gfCNCPoint3[21625] = {X 108.1088, Y 46.8612, Z -4.6667, A 0.000, B 0.000, C 0.000 }
gfCNCPoint3[21626] = {X 107.7913, Y 45.9714, Z -4.6667, A 0.000, B 0.000, C 0.000 }
gfCNCPoint3[21627] = {X 107.6786, Y 45.0335, Z -4.6667, A 0.000, B 0.000, C 0.000 }
gfCNCPoint3[21628] = {X 107.6785, Y 44.1775, Z -4.6667, A 0.000, B 0.000, C 0.000 }
gfCNCPoint3[21629] = {X 107.7133, Y 43.6465, Z -4.6667, A 0.000, B 0.000, C 0.000 }
gfCNCPoint3[21630] = {X 107.8171, Y 43.1246, Z -4.6667, A 0.000, B 0.000, C 0.000 }
gfCNCPoint3[21631] = {X 107.9815, Y 42.6369, Z -4.6667, A 0.000, B 0.000, C 0.000 }
gfCNCPoint3[21632] = {X 108.2062, Y 42.1739, Z -4.6667, A 0.000, B 0.000, C 0.000 }
gfCNCPoint3[21633] = {X 108.6606, Y 41.4995, Z -4.6667, A 0.000, B 0.000, C 0.000 }
gfCNCPoint3[21634] = {X 109.2059, Y 40.8963, Z -4.6667, A 0.000, B 0.000, C 0.000 }
gfCNCPoint3[21635] = {X 109.2058, Y 39.1629, Z -4.6667, A 0.000, B 0.000, C 0.000 }
gfCNCPoint3[21636] = {X 109.0939, Y 39.1629, Z -4.6667, A 0.000, B 0.000, C 0.000 }
gfCNCPoint3[21637] = {X 106.0379, Y 46.6307, Z -4.6667, A 0.000, B 0.000, C 0.000 }
gfCNCPoint3[21638] = {X 105.6747, Y 47.3174, Z -4.6667, A 0.000, B 0.000, C 0.000 }
gfCNCPoint3[21639] = {X 105.1923, Y 47.9263, Z -4.6667, A 0.000, B 0.000, C 0.000 }
gfCNCPoint3[21640] = {X 104.6069, Y 48.4370, Z -4.6667, A 0.000, B 0.000, C 0.000 }
gfCNCPoint3[21641] = {X 103.9382, Y 48.8323, Z -4.6667, A 0.000, B 0.000, C 0.000 }
gfCNCPoint3[21642] = {X 103.0119, Y 49.1460, Z -4.6667, A 0.000, B 0.000, C 0.000 }
gfCNCPoint3[21643] = {X 102.0384, Y 49.2391, Z -4.6667, A 0.000, B 0.000, C 0.000 }
gfCNCPoint3[21644] = {X 101.0695, Y 49.1068, Z -4.6667, A 0.000, B 0.000, C 0.000 }
gfCNCPoint3[21645] = {X 100.1566, Y 48.7559, Z -4.6667, A 0.000, B 0.000, C 0.000 }
gfCNCPoint3[21646] = {X 99.3484, Y 48.2052, Z -4.6667, A 0.000, B 0.000, C 0.000 }
gfCNCPoint3[21647] = {X 98.6879, Y 47.4840, Z -4.6667, A 0.000, B 0.000, C 0.000 }
gfCNCPoint3[21648] = {X 98.2102, Y 46.6307, Z -4.6667, A 0.000, B 0.000, C 0.000 }
gfCNCPoint3[21649] = {X 95.0510, Y 38.9046, Z -4.6667, A 0.000, B 0.000, C 0.000 }
gfCNCPoint3[21650] = {X 95.0511, Y 40.9419, Z -4.6667, A 0.000, B 0.000, C 0.000 }
gfCNCPoint3[21651] = {X 95.5851, Y 41.4821, Z -4.6667, A 0.000, B 0.000, C 0.000 }
gfCNCPoint3[21652] = {X 96.0162, Y 42.1073, Z -4.6667, A 0.000, B 0.000, C 0.000 }
gfCNCPoint3[21653] = {X 96.2570, Y 42.6034, Z -4.6667, A 0.000, B 0.000, C 0.000 }
gfCNCPoint3[21654] = {X 96.4328, Y 43.1260, Z -4.6667, A 0.000, B 0.000, C 0.000 }
gfCNCPoint3[21655] = {X 96.5399, Y 43.6619, Z -4.6667, A 0.000, B 0.000, C 0.000 }
gfCNCPoint3[21656] = {X 96.5785, Y 44.2071, Z -4.6667, A 0.000, B 0.000, C 0.000 }
gfCNCPoint3[21657] = {X 96.5783, Y 45.0408, Z -4.6667, A 0.000, B 0.000, C 0.000 }
gfCNCPoint3[21658] = {X 96.4643, Y 45.9775, Z -4.6667, A 0.000, B 0.000, C 0.000 }
gfCNCPoint3[21659] = {X 96.1459, Y 46.8659, Z -4.6667, A 0.000, B 0.000, C 0.000 }
gfCNCPoint3[21660] = {X 95.6389, Y 47.6618, Z -4.6667, A 0.000, B 0.000, C 0.000 }
gfCNCPoint3[21661] = {X 94.9685, Y 48.3258, Z -4.6667, A 0.000, B 0.000, C 0.000 }
gfCNCPoint3[21662] = {X 94.1677, Y 48.8251, Z -4.6667, A 0.000, B 0.000, C 0.000 }
gfCNCPoint3[21663] = {X 93.2764, Y 49.1350, Z -4.6667, A 0.000, B 0.000, C 0.000 }
gfCNCPoint3[21664] = {X 92.3385, Y 49.2400, Z -4.6667, A 0.000, B 0.000, C 0.000 }
gfCNCPoint3[21665] = {X 85.8951, Y 49.2400, Z -4.6667, A 0.000, B 0.000, C 0.000 }
gfCNCPoint3[21666] = {X 84.9564, Y 49.1348, Z -4.6667, A 0.000, B 0.000, C 0.000 }
gfCNCPoint3[21667] = {X 84.0643, Y 48.8244, Z -4.6667, A 0.000, B 0.000, C 0.000 }
gfCNCPoint3[21668] = {X 83.2631, Y 48.3242, Z -4.6667, A 0.000, B 0.000, C 0.000 }
gfCNCPoint3[21669] = {X 82.5924, Y 47.6590, Z -4.6667, A 0.000, B 0.000, C 0.000 }
gfCNCPoint3[21670] = {X 82.0857, Y 46.8618, Z -4.6667, A 0.000, B 0.000, C 0.000 }
gfCNCPoint3[21671] = {X 81.7681, Y 45.9723, Z -4.6667, A 0.000, B 0.000, C 0.000 }
gfCNCPoint3[21672] = {X 81.6552, Y 45.0345, Z -4.6667, A 0.000, B 0.000, C 0.000 }
gfCNCPoint3[21673] = {X 81.6551, Y 44.2075, Z -4.6667, A 0.000, B 0.000, C 0.000 }
gfCNCPoint3[21674] = {X 81.7604, Y 43.2862, Z -4.6667, A 0.000, B 0.000, C 0.000 }
gfCNCPoint3[21675] = {X 82.0609, Y 42.4090, Z -4.6667, A 0.000, B 0.000, C 0.000 }
gfCNCPoint3[21676] = {X 82.5425, Y 41.6167, Z -4.6667, A 0.000, B 0.000, C 0.000 }
gfCNCPoint3[21677] = {X 83.1828, Y 40.9460, Z -4.6667, A 0.000, B 0.000, C 0.000 }
gfCNCPoint3[21678] = {X 83.1826, Y 28.5916, Z -4.6667, A 0.000, B 0.000, C 0.000 }
gfCNCPoint3[21679] = {X 79.1826, Y 28.5916, Z -4.6667, A 0.000, B 0.000, C 0.000 }
gfCNCPoint3[21680] = {X 83.2626, Y 28.5916, Z -4.6667, A 0.000, B 0.000, C 0.000 }
gfCNCPoint3[21681] = {X 83.2625, Y 16.1991, Z -4.6667, A 0.000, B 0.000, C 0.000 }
gfCNCPoint3[21682] = {X 82.6249, Y 15.5494, Z -4.6667, A 0.000, B 0.000, C 0.000 }
gfCNCPoint3[21683] = {X 82.1439, Y 14.7765, Z -4.6667, A 0.000, B 0.000, C 0.000 }
gfCNCPoint3[21684] = {X 81.8426, Y 13.9176, Z -4.6667, A 0.000, B 0.000, C 0.000 }
gfCNCPoint3[21685] = {X 81.7352, Y 13.0136, Z -4.6667, A 0.000, B 0.000, C 0.000 }
gfCNCPoint3[21686] = {X 81.7351, Y 12.1868, Z -4.6667, A 0.000, B 0.000, C 0.000 }
gfCNCPoint3[21687] = {X 81.8394, Y 11.2611, Z -4.6667, A 0.000, B 0.000, C 0.000 }
gfCNCPoint3[21688] = {X 82.1470, Y 10.3819, Z -4.6667, A 0.000, B 0.000, C 0.000 }
gfCNCPoint3[21689] = {X 82.6427, Y 9.5931, Z -4.6667, A 0.000, B 0.000, C 0.000 }
gfCNCPoint3[21690] = {X 83.3014, Y 8.9344, Z -4.6667, A 0.000, B 0.000, C 0.000 }
gfCNCPoint3[21691] = {X 84.0901, Y 8.4388, Z -4.6667, A 0.000, B 0.000, C 0.000 }
gfCNCPoint3[21692] = {X 84.9694, Y 8.1311, Z -4.6667, A 0.000, B 0.000, C 0.000 }
gfCNCPoint3[21693] = {X 85.8951, Y 8.0268, Z -4.6667, A 0.000, B 0.000, C 0.000 }
gfCNCPoint3[21694] = {X 94.0497, Y 8.0268, Z -4.6667, A 0.000, B 0.000, C 0.000 }
gfCNCPoint3[21695] = {X 94.9754, Y 8.1311, Z -4.6667, A 0.000, B 0.000, C 0.000 }
gfCNCPoint3[21696] = {X 95.8546, Y 8.4388, Z -4.6667, A 0.000, B 0.000, C 0.000 }
gfCNCPoint3[21697] = {X 96.6434, Y 8.9344, Z -4.6667, A 0.000, B 0.000, C 0.000 }
gfCNCPoint3[21698] = {X 97.3021, Y 9.5931, Z -4.6667, A 0.000, B 0.000, C 0.000 }
gfCNCPoint3[21699] = {X 97.7977, Y 10.3819, Z -4.6667, A 0.000, B 0.000, C 0.000 }
gfCNCPoint3[21700] = {X 98.1054, Y 11.2611, Z -4.6667, A 0.000, B 0.000, C 0.000 }
gfCNCPoint3[21701] = {X 98.2097, Y 12.1868, Z -4.6667, A 0.000, B 0.000, C 0.000 }
gfCNCPoint3[21702] = {X 98.2097, Y 12.9782, Z -4.6667, A 0.000, B 0.000, C 0.000 }
gfCNCPoint3[21703] = {X 98.1344, Y 13.7659, Z -4.6667, A 0.000, B 0.000, C 0.000 }
gfCNCPoint3[21704] = {X 97.9112, Y 14.5252, Z -4.6667, A 0.000, B 0.000, C 0.000 }
gfCNCPoint3[21705] = {X 97.5484, Y 15.2285, Z -4.6667, A 0.000, B 0.000, C 0.000 }
gfCNCPoint3[21706] = {X 101.8773, Y 25.9551, Z -4.6667, A 0.000, B 0.000, C 0.000 }
gfCNCPoint3[21707] = {X 101.9779, Y 25.7088, Z -4.6667, A 0.000, B 0.000, C 0.000 }
gfCNCPoint3[21708] = {X 106.1951, Y 15.2059, Z -4.6667, A 0.000, B 0.000, C 0.000 }
gfCNCPoint3[21709] = {X 105.8448, Y 14.5204, Z -4.6667, A 0.000, B 0.000, C 0.000 }
gfCNCPoint3[21710] = {X 105.6267, Y 13.7822, Z -4.6667, A 0.000, B 0.000, C 0.000 }
gfCNCPoint3[21711] = {X 105.5485, Y 13.0164, Z -4.6667, A 0.000, B 0.000, C 0.000 }
gfCNCPoint3[21712] = {X 105.5483, Y 12.1868, Z -4.6667, A 0.000, B 0.000, C 0.000 }
gfCNCPoint3[21713] = {X 105.6526, Y 11.2611, Z -4.6667, A 0.000, B 0.000, C 0.000 }
gfCNCPoint3[21714] = {X 105.9602, Y 10.3819, Z -4.6667, A 0.000, B 0.000, C 0.000 }
gfCNCPoint3[21715] = {X 106.4559, Y 9.5931, Z -4.6667, A 0.000, B 0.000, C 0.000 }
gfCNCPoint3[21716] = {X 107.1146, Y 8.9344, Z -4.6667, A 0.000, B 0.000, C 0.000 }
gfCNCPoint3[21717] = {X 107.9033, Y 8.4388, Z -4.6667, A 0.000, B 0.000, C 0.000 }
gfCNCPoint3[21718] = {X 108.7826, Y 8.1311, Z -4.6667, A 0.000, B 0.000, C 0.000 }
gfCNCPoint3[21719] = {X 109.7083, Y 8.0268, Z -4.6667, A 0.000, B 0.000, C 0.000 }
gfCNCPoint3[21720] = {X 117.7916, Y 8.0268, Z -4.6667, A 0.000, B 0.000, C 0.000 }
gfCNCPoint3[21721] = {X 118.7173, Y 8.1311, Z -4.6667, A 0.000, B 0.000, C 0.000 }
gfCNCPoint3[21722] = {X 119.5965, Y 8.4388, Z -4.6667, A 0.000, B 0.000, C 0.000 }
gfCNCPoint3[21723] = {X 120.3853, Y 8.9344, Z -4.6667, A 0.000, B 0.000, C 0.000 }
gfCNCPoint3[21724] = {X 121.0440, Y 9.5931, Z -4.6667, A 0.000, B 0.000, C 0.000 }
gfCNCPoint3[21725] = {X 121.5396, Y 10.3819, Z -4.6667, A 0.000, B 0.000, C 0.000 }
gfCNCPoint3[21726] = {X 121.8473, Y 11.2611, Z -4.6667, A 0.000, B 0.000, C 0.000 }
gfCNCPoint3[21727] = {X 121.9516, Y 12.1868, Z -4.6667, A 0.000, B 0.000, C 0.000 }
gfCNCPoint3[21728] = {X 121.9516, Y 12.9782, Z -4.6667, A 0.000, B 0.000, C 0.000 }
gfCNCPoint3[21729] = {X 121.8501, Y 13.8913, Z -4.6667, A 0.000, B 0.000, C 0.000 }
gfCNCPoint3[21730] = {X 121.5506, Y 14.7599, Z -4.6667, A 0.000, B 0.000, C 0.000 }
gfCNCPoint3[21731] = {X 121.0678, Y 15.5416, Z -4.6667, A 0.000, B 0.000, C 0.000 }
gfCNCPoint3[21732] = {X 120.4251, Y 16.1983, Z -4.6667, A 0.000, B 0.000, C 0.000 }
gfCNCPoint3[21733] = {X 120.4241, Y 40.9900, Z -4.6667, A 0.000, B 0.000, C 0.000 }
gfCNCPoint3[21734] = {X 120.5191, Y 41.0678, Z -4.6667, A 0.000, B 0.000, C 0.000 }
gfCNCPoint3[21735] = {X 121.1187, Y 41.7116, Z -4.6667, A 0.000, B 0.000, C 0.000 }
gfCNCPoint3[21736] = {X 121.5695, Y 42.4672, Z -4.6667, A 0.000, B 0.000, C 0.000 }
gfCNCPoint3[21737] = {X 121.8512, Y 43.3006, Z -4.6667, A 0.000, B 0.000, C 0.000 }
gfCNCPoint3[21738] = {X 121.9514, Y 44.1747, Z -4.6667, A 0.000, B 0.000, C 0.000 }
gfCNCPoint3[21739] = {X 121.9516, Y 45.0000, Z -4.6667, A 0.000, B 0.000, C 0.000 }
gfCNCPoint3[21740] = {X 121.8473, Y 45.9257, Z -4.6667, A 0.000, B 0.000, C 0.000 }
gfCNCPoint3[21741] = {X 121.5396, Y 46.8050, Z -4.6667, A 0.000, B 0.000, C 0.000 }
gfCNCPoint3[21742] = {X 121.0440, Y 47.5937, Z -4.6667, A 0.000, B 0.000, C 0.000 }
gfCNCPoint3[21743] = {X 120.3853, Y 48.2524, Z -4.6667, A 0.000, B 0.000, C 0.000 }
gfCNCPoint3[21744] = {X 119.5965, Y 48.7480, Z -4.6667, A 0.000, B 0.000, C 0.000 }
gfCNCPoint3[21745] = {X 118.7173, Y 49.0557, Z -4.6667, A 0.000, B 0.000, C 0.000 }
gfCNCPoint3[21746] = {X 117.7916, Y 49.1600, Z -4.6667, A 0.000, B 0.000, C 0.000 }
gfCNCPoint3[21747] = {X 111.9185, Y 49.1600, Z -4.6667, A 0.000, B 0.000, C 0.000 }
gfCNCPoint3[21748] = {X 110.9974, Y 49.0567, Z -4.6667, A 0.000, B 0.000, C 0.000 }
gfCNCPoint3[21749] = {X 110.1220, Y 48.7521, Z -4.6667, A 0.000, B 0.000, C 0.000 }
gfCNCPoint3[21750] = {X 109.3358, Y 48.2612, Z -4.6667, A 0.000, B 0.000, C 0.000 }
gfCNCPoint3[21751] = {X 108.6778, Y 47.6084, Z -4.6667, A 0.000, B 0.000, C 0.000 }
gfCNCPoint3[21752] = {X 108.1807, Y 46.8261, Z -4.6667, A 0.000, B 0.000, C 0.000 }
gfCNCPoint3[21753] = {X 107.8691, Y 45.9531, Z -4.6667, A 0.000, B 0.000, C 0.000 }
gfCNCPoint3[21754] = {X 107.7586, Y 45.0328, Z -4.6667, A 0.000, B 0.000, C 0.000 }
gfCNCPoint3[21755] = {X 107.7585, Y 44.1775, Z -4.6667, A 0.000, B 0.000, C 0.000 }
gfCNCPoint3[21756] = {X 107.7926, Y 43.6570, Z -4.6667, A 0.000, B 0.000, C 0.000 }
gfCNCPoint3[21757] = {X 107.8944, Y 43.1453, Z -4.6667, A 0.000, B 0.000, C 0.000 }
gfCNCPoint3[21758] = {X 108.0555, Y 42.6672, Z -4.6667, A 0.000, B 0.000, C 0.000 }
gfCNCPoint3[21759] = {X 108.2758, Y 42.2133, Z -4.6667, A 0.000, B 0.000, C 0.000 }
gfCNCPoint3[21760] = {X 108.7343, Y 41.5352, Z -4.6667, A 0.000, B 0.000, C 0.000 }
gfCNCPoint3[21761] = {X 109.2859, Y 40.9305, Z -4.6667, A 0.000, B 0.000, C 0.000 }
gfCNCPoint3[21762] = {X 109.2858, Y 39.0829, Z -4.6667, A 0.000, B 0.000, C 0.000 }
gfCNCPoint3[21763] = {X 109.0402, Y 39.0829, Z -4.6667, A 0.000, B 0.000, C 0.000 }
gfCNCPoint3[21764] = {X 105.9641, Y 46.5999, Z -4.6667, A 0.000, B 0.000, C 0.000 }
gfCNCPoint3[21765] = {X 105.6077, Y 47.2737, Z -4.6667, A 0.000, B 0.000, C 0.000 }
gfCNCPoint3[21766] = {X 105.1344, Y 47.8711, Z -4.6667, A 0.000, B 0.000, C 0.000 }
gfCNCPoint3[21767] = {X 104.5601, Y 48.3721, Z -4.6667, A 0.000, B 0.000, C 0.000 }
gfCNCPoint3[21768] = {X 103.9040, Y 48.7600, Z -4.6667, A 0.000, B 0.000, C 0.000 }
gfCNCPoint3[21769] = {X 102.9952, Y 49.0678, Z -4.6667, A 0.000, B 0.000, C 0.000 }
gfCNCPoint3[21770] = {X 102.0400, Y 49.1592, Z -4.6667, A 0.000, B 0.000, C 0.000 }
gfCNCPoint3[21771] = {X 101.0894, Y 49.0293, Z -4.6667, A 0.000, B 0.000, C 0.000 }
gfCNCPoint3[21772] = {X 100.1937, Y 48.6850, Z -4.6667, A 0.000, B 0.000, C 0.000 }
gfCNCPoint3[21773] = {X 99.4008, Y 48.1448, Z -4.6667, A 0.000, B 0.000, C 0.000 }
gfCNCPoint3[21774] = {X 98.7527, Y 47.4372, Z -4.6667, A 0.000, B 0.000, C 0.000 }
gfCNCPoint3[21775] = {X 98.2840, Y 46.5999, Z -4.6667, A 0.000, B 0.000, C 0.000 }
gfCNCPoint3[21776] = {X 94.9710, Y 38.4975, Z -4.6667, A 0.000, B 0.000, C 0.000 }
gfCNCPoint3[21777] = {X 94.9711, Y 40.9792, Z -4.6667, A 0.000, B 0.000, C 0.000 }
gfCNCPoint3[21778] = {X 95.5116, Y 41.5189, Z -4.6667, A 0.000, B 0.000, C 0.000 }
gfCNCPoint3[21779] = {X 95.9466, Y 42.1468, Z -4.6667, A 0.000, B 0.000, C 0.000 }
gfCNCPoint3[21780] = {X 96.1830, Y 42.6336, Z -4.6667, A 0.000, B 0.000, C 0.000 }
gfCNCPoint3[21781] = {X 96.3555, Y 43.1466, Z -4.6667, A 0.000, B 0.000, C 0.000 }
gfCNCPoint3[21782] = {X 96.4606, Y 43.6726, Z -4.6667, A 0.000, B 0.000, C 0.000 }
gfCNCPoint3[21783] = {X 96.4985, Y 44.2077, Z -4.6667, A 0.000, B 0.000, C 0.000 }
gfCNCPoint3[21784] = {X 96.4983, Y 45.0400, Z -4.6667, A 0.000, B 0.000, C 0.000 }
gfCNCPoint3[21785] = {X 96.3865, Y 45.9591, Z -4.6667, A 0.000, B 0.000, C 0.000 }
gfCNCPoint3[21786] = {X 96.0741, Y 46.8306, Z -4.6667, A 0.000, B 0.000, C 0.000 }
gfCNCPoint3[21787] = {X 95.5767, Y 47.6115, Z -4.6667, A 0.000, B 0.000, C 0.000 }
gfCNCPoint3[21788] = {X 94.9188, Y 48.2631, Z -4.6667, A 0.000, B 0.000, C 0.000 }
gfCNCPoint3[21789] = {X 94.1332, Y 48.7530, Z -4.6667, A 0.000, B 0.000, C 0.000 }
gfCNCPoint3[21790] = {X 93.2587, Y 49.0570, Z -4.6667, A 0.000, B 0.000, C 0.000 }
gfCNCPoint3[21791] = {X 92.3385, Y 49.1600, Z -4.6667, A 0.000, B 0.000, C 0.000 }
gfCNCPoint3[21792] = {X 85.8951, Y 49.1600, Z -4.6667, A 0.000, B 0.000, C 0.000 }
gfCNCPoint3[21793] = {X 84.9741, Y 49.0568, Z -4.6667, A 0.000, B 0.000, C 0.000 }
gfCNCPoint3[21794] = {X 84.0988, Y 48.7522, Z -4.6667, A 0.000, B 0.000, C 0.000 }
gfCNCPoint3[21795] = {X 83.3127, Y 48.2614, Z -4.6667, A 0.000, B 0.000, C 0.000 }
gfCNCPoint3[21796] = {X 82.6547, Y 47.6088, Z -4.6667, A 0.000, B 0.000, C 0.000 }
gfCNCPoint3[21797] = {X 82.1576, Y 46.8267, Z -4.6667, A 0.000, B 0.000, C 0.000 }
gfCNCPoint3[21798] = {X 81.8459, Y 45.9539, Z -4.6667, A 0.000, B 0.000, C 0.000 }
gfCNCPoint3[21799] = {X 81.7352, Y 45.0338, Z -4.6667, A 0.000, B 0.000, C 0.000 }
gfCNCPoint3[21800] = {X 81.7351, Y 44.2079, Z -4.6667, A 0.000, B 0.000, C 0.000 }
gfCNCPoint3[21801] = {X 81.8405, Y 43.2948, Z -4.6667, A 0.000, B 0.000, C 0.000 }
gfCNCPoint3[21802] = {X 82.1412, Y 42.4262, Z -4.6667, A 0.000, B 0.000, C 0.000 }
gfCNCPoint3[21803] = {X 82.6229, Y 41.6434, Z -4.6667, A 0.000, B 0.000, C 0.000 }
gfCNCPoint3[21804] = {X 83.2628, Y 40.9834, Z -4.6667, A 0.000, B 0.000, C 0.000 }
gfCNCPoint3[21805] = {X 83.2626, Y 28.5916, Z -4.6667, A 0.000, B 0.000, C 0.000 }
gfCNCPoint3[21806] = {X 79.2626, Y 28.5916, Z -4.6667, A 0.000, B 0.000, C 0.000 }
gfCNCPoint3[21807] = {X 83.3426, Y 28.5916, Z -4.6667, A 0.000, B 0.000, C 0.000 }
gfCNCPoint3[21808] = {X 83.3425, Y 16.1609, Z -4.6667, A 0.000, B 0.000, C 0.000 }
gfCNCPoint3[21809] = {X 82.7054, Y 15.5221, Z -4.6667, A 0.000, B 0.000, C 0.000 }
gfCNCPoint3[21810] = {X 82.2243, Y 14.7589, Z -4.6667, A 0.000, B 0.000, C 0.000 }
gfCNCPoint3[21811] = {X 81.9226, Y 13.9087, Z -4.6667, A 0.000, B 0.000, C 0.000 }
gfCNCPoint3[21812] = {X 81.8152, Y 13.0129, Z -4.6667, A 0.000, B 0.000, C 0.000 }
gfCNCPoint3[21813] = {X 81.8151, Y 12.1868, Z -4.6667, A 0.000, B 0.000, C 0.000 }
gfCNCPoint3[21814] = {X 81.9174, Y 11.2789, Z -4.6667, A 0.000, B 0.000, C 0.000 }
gfCNCPoint3[21815] = {X 82.2191, Y 10.4166, Z -4.6667, A 0.000, B 0.000, C 0.000 }
gfCNCPoint3[21816] = {X 82.7052, Y 9.6430, Z -4.6667, A 0.000, B 0.000, C 0.000 }
gfCNCPoint3[21817] = {X 83.3512, Y 8.9969, Z -4.6667, A 0.000, B 0.000, C 0.000 }
gfCNCPoint3[21818] = {X 84.1248, Y 8.5109, Z -4.6667, A 0.000, B 0.000, C 0.000 }
gfCNCPoint3[21819] = {X 84.9872, Y 8.2091, Z -4.6667, A 0.000, B 0.000, C 0.000 }
gfCNCPoint3[21820] = {X 85.8951, Y 8.1068, Z -4.6667, A 0.000, B 0.000, C 0.000 }
gfCNCPoint3[21821] = {X 94.0497, Y 8.1068, Z -4.6667, A 0.000, B 0.000, C 0.000 }
gfCNCPoint3[21822] = {X 94.9576, Y 8.2091, Z -4.6667, A 0.000, B 0.000, C 0.000 }
gfCNCPoint3[21823] = {X 95.8199, Y 8.5109, Z -4.6667, A 0.000, B 0.000, C 0.000 }
gfCNCPoint3[21824] = {X 96.5935, Y 8.9969, Z -4.6667, A 0.000, B 0.000, C 0.000 }
gfCNCPoint3[21825] = {X 97.2395, Y 9.6430, Z -4.6667, A 0.000, B 0.000, C 0.000 }
gfCNCPoint3[21826] = {X 97.7256, Y 10.4166, Z -4.6667, A 0.000, B 0.000, C 0.000 }
gfCNCPoint3[21827] = {X 98.0274, Y 11.2789, Z -4.6667, A 0.000, B 0.000, C 0.000 }
gfCNCPoint3[21828] = {X 98.1297, Y 12.1868, Z -4.6667, A 0.000, B 0.000, C 0.000 }
gfCNCPoint3[21829] = {X 98.1297, Y 12.9782, Z -4.6667, A 0.000, B 0.000, C 0.000 }
gfCNCPoint3[21830] = {X 98.0631, Y 13.7120, Z -4.6667, A 0.000, B 0.000, C 0.000 }
gfCNCPoint3[21831] = {X 97.8656, Y 14.4219, Z -4.6667, A 0.000, B 0.000, C 0.000 }
gfCNCPoint3[21832] = {X 97.5437, Y 15.0847, Z -4.6667, A 0.000, B 0.000, C 0.000 }
gfCNCPoint3[21833] = {X 97.4973, Y 15.1598, Z -4.6667, A 0.000, B 0.000, C 0.000 }
gfCNCPoint3[21834] = {X 97.4492, Y 15.2340, Z -4.6667, A 0.000, B 0.000, C 0.000 }
gfCNCPoint3[21835] = {X 97.4854, Y 15.2810, Z -4.6667, A 0.000, B 0.000, C 0.000 }
gfCNCPoint3[21836] = {X 101.8768, Y 26.1678, Z -4.6667, A 0.000, B 0.000, C 0.000 }
gfCNCPoint3[21837] = {X 102.0520, Y 25.7389, Z -4.6667, A 0.000, B 0.000, C 0.000 }
gfCNCPoint3[21838] = {X 106.2847, Y 15.1974, Z -4.6667, A 0.000, B 0.000, C 0.000 }
gfCNCPoint3[21839] = {X 106.2413, Y 15.1289, Z -4.6667, A 0.000, B 0.000, C 0.000 }
gfCNCPoint3[21840] = {X 106.1992, Y 15.0596, Z -4.6667, A 0.000, B 0.000, C 0.000 }
gfCNCPoint3[21841] = {X 105.8898, Y 14.4153, Z -4.6667, A 0.000, B 0.000, C 0.000 }
gfCNCPoint3[21842] = {X 105.6976, Y 13.7270, Z -4.6667, A 0.000, B 0.000, C 0.000 }
gfCNCPoint3[21843] = {X 105.6285, Y 13.0157, Z -4.6667, A 0.000, B 0.000, C 0.000 }
gfCNCPoint3[21844] = {X 105.6283, Y 12.1868, Z -4.6667, A 0.000, B 0.000, C 0.000 }
gfCNCPoint3[21845] = {X 105.7306, Y 11.2789, Z -4.6667, A 0.000, B 0.000, C 0.000 }
gfCNCPoint3[21846] = {X 106.0323, Y 10.4166, Z -4.6667, A 0.000, B 0.000, C 0.000 }
gfCNCPoint3[21847] = {X 106.5184, Y 9.6430, Z -4.6667, A 0.000, B 0.000, C 0.000 }
gfCNCPoint3[21848] = {X 107.1644, Y 8.9969, Z -4.6667, A 0.000, B 0.000, C 0.000 }
gfCNCPoint3[21849] = {X 107.9380, Y 8.5109, Z -4.6667, A 0.000, B 0.000, C 0.000 }
gfCNCPoint3[21850] = {X 108.8004, Y 8.2091, Z -4.6667, A 0.000, B 0.000, C 0.000 }
gfCNCPoint3[21851] = {X 109.7083, Y 8.1068, Z -4.6667, A 0.000, B 0.000, C 0.000 }
gfCNCPoint3[21852] = {X 117.7916, Y 8.1068, Z -4.6667, A 0.000, B 0.000, C 0.000 }
gfCNCPoint3[21853] = {X 118.6995, Y 8.2091, Z -4.6667, A 0.000, B 0.000, C 0.000 }
gfCNCPoint3[21854] = {X 119.5618, Y 8.5109, Z -4.6667, A 0.000, B 0.000, C 0.000 }
gfCNCPoint3[21855] = {X 120.3354, Y 8.9969, Z -4.6667, A 0.000, B 0.000, C 0.000 }
gfCNCPoint3[21856] = {X 120.9814, Y 9.6430, Z -4.6667, A 0.000, B 0.000, C 0.000 }
gfCNCPoint3[21857] = {X 121.4675, Y 10.4166, Z -4.6667, A 0.000, B 0.000, C 0.000 }
gfCNCPoint3[21858] = {X 121.7693, Y 11.2789, Z -4.6667, A 0.000, B 0.000, C 0.000 }
gfCNCPoint3[21859] = {X 121.8716, Y 12.1868, Z -4.6667, A 0.000, B 0.000, C 0.000 }
gfCNCPoint3[21860] = {X 121.8716, Y 12.9782, Z -4.6667, A 0.000, B 0.000, C 0.000 }
gfCNCPoint3[21861] = {X 121.7700, Y 13.8830, Z -4.6667, A 0.000, B 0.000, C 0.000 }
gfCNCPoint3[21862] = {X 121.4702, Y 14.7427, Z -4.6667, A 0.000, B 0.000, C 0.000 }
gfCNCPoint3[21863] = {X 120.9872, Y 15.5146, Z -4.6667, A 0.000, B 0.000, C 0.000 }
gfCNCPoint3[21864] = {X 120.3451, Y 16.1601, Z -4.6667, A 0.000, B 0.000, C 0.000 }
gfCNCPoint3[21865] = {X 120.3441, Y 41.0280, Z -4.6667, A 0.000, B 0.000, C 0.000 }
gfCNCPoint3[21866] = {X 120.4676, Y 41.1289, Z -4.6667, A 0.000, B 0.000, C 0.000 }
gfCNCPoint3[21867] = {X 121.0552, Y 41.7604, Z -4.6667, A 0.000, B 0.000, C 0.000 }
gfCNCPoint3[21868] = {X 121.4971, Y 42.5012, Z -4.6667, A 0.000, B 0.000, C 0.000 }
gfCNCPoint3[21869] = {X 121.7732, Y 43.3184, Z -4.6667, A 0.000, B 0.000, C 0.000 }
gfCNCPoint3[21870] = {X 121.8714, Y 44.1754, Z -4.6667, A 0.000, B 0.000, C 0.000 }
gfCNCPoint3[21871] = {X 121.8716, Y 45.0000, Z -4.6667, A 0.000, B 0.000, C 0.000 }
gfCNCPoint3[21872] = {X 121.7693, Y 45.9079, Z -4.6667, A 0.000, B 0.000, C 0.000 }
gfCNCPoint3[21873] = {X 121.4675, Y 46.7702, Z -4.6667, A 0.000, B 0.000, C 0.000 }
gfCNCPoint3[21874] = {X 120.9814, Y 47.5438, Z -4.6667, A 0.000, B 0.000, C 0.000 }
gfCNCPoint3[21875] = {X 120.3354, Y 48.1899, Z -4.6667, A 0.000, B 0.000, C 0.000 }
gfCNCPoint3[21876] = {X 119.5618, Y 48.6760, Z -4.6667, A 0.000, B 0.000, C 0.000 }
gfCNCPoint3[21877] = {X 118.6995, Y 48.9777, Z -4.6667, A 0.000, B 0.000, C 0.000 }
gfCNCPoint3[21878] = {X 117.7916, Y 49.0800, Z -4.6667, A 0.000, B 0.000, C 0.000 }
gfCNCPoint3[21879] = {X 111.9185, Y 49.0800, Z -4.6667, A 0.000, B 0.000, C 0.000 }
gfCNCPoint3[21880] = {X 111.0151, Y 48.9787, Z -4.6667, A 0.000, B 0.000, C 0.000 }
gfCNCPoint3[21881] = {X 110.1565, Y 48.6799, Z -4.6667, A 0.000, B 0.000, C 0.000 }
gfCNCPoint3[21882] = {X 109.3855, Y 48.1985, Z -4.6667, A 0.000, B 0.000, C 0.000 }
gfCNCPoint3[21883] = {X 108.7401, Y 47.5582, Z -4.6667, A 0.000, B 0.000, C 0.000 }
gfCNCPoint3[21884] = {X 108.2526, Y 46.7909, Z -4.6667, A 0.000, B 0.000, C 0.000 }
gfCNCPoint3[21885] = {X 107.9470, Y 45.9348, Z -4.6667, A 0.000, B 0.000, C 0.000 }
gfCNCPoint3[21886] = {X 107.8386, Y 45.0322, Z -4.6667, A 0.000, B 0.000, C 0.000 }
gfCNCPoint3[21887] = {X 107.8385, Y 44.1775, Z -4.6667, A 0.000, B 0.000, C 0.000 }
gfCNCPoint3[21888] = {X 107.8719, Y 43.6674, Z -4.6667, A 0.000, B 0.000, C 0.000 }
gfCNCPoint3[21889] = {X 107.9716, Y 43.1661, Z -4.6667, A 0.000, B 0.000, C 0.000 }
gfCNCPoint3[21890] = {X 108.1296, Y 42.6975, Z -4.6667, A 0.000, B 0.000, C 0.000 }
gfCNCPoint3[21891] = {X 108.3454, Y 42.2527, Z -4.6667, A 0.000, B 0.000, C 0.000 }
gfCNCPoint3[21892] = {X 108.8080, Y 41.5711, Z -4.6667, A 0.000, B 0.000, C 0.000 }
gfCNCPoint3[21893] = {X 109.3659, Y 40.9650, Z -4.6667, A 0.000, B 0.000, C 0.000 }
gfCNCPoint3[21894] = {X 109.3658, Y 39.0029, Z -4.6667, A 0.000, B 0.000, C 0.000 }
gfCNCPoint3[21895] = {X 108.9865, Y 39.0029, Z -4.6667, A 0.000, B 0.000, C 0.000 }
gfCNCPoint3[21896] = {X 105.8902, Y 46.5692, Z -4.6667, A 0.000, B 0.000, C 0.000 }
gfCNCPoint3[21897] = {X 105.5407, Y 47.2300, Z -4.6667, A 0.000, B 0.000, C 0.000 }
gfCNCPoint3[21898] = {X 105.0765, Y 47.8159, Z -4.6667, A 0.000, B 0.000, C 0.000 }
gfCNCPoint3[21899] = {X 104.5133, Y 48.3073, Z -4.6667, A 0.000, B 0.000, C 0.000 }
gfCNCPoint3[21900] = {X 103.8698, Y 48.6877, Z -4.6667, A 0.000, B 0.000, C 0.000 }
gfCNCPoint3[21901] = {X 102.9784, Y 48.9895, Z -4.6667, A 0.000, B 0.000, C 0.000 }
gfCNCPoint3[21902] = {X 102.0417, Y 49.0792, Z -4.6667, A 0.000, B 0.000, C 0.000 }
gfCNCPoint3[21903] = {X 101.1093, Y 48.9518, Z -4.6667, A 0.000, B 0.000, C 0.000 }
gfCNCPoint3[21904] = {X 100.2309, Y 48.6142, Z -4.6667, A 0.000, B 0.000, C 0.000 }
gfCNCPoint3[21905] = {X 99.4532, Y 48.0843, Z -4.6667, A 0.000, B 0.000, C 0.000 }
gfCNCPoint3[21906] = {X 98.8176, Y 47.3903, Z -4.6667, A 0.000, B 0.000, C 0.000 }
gfCNCPoint3[21907] = {X 98.3579, Y 46.5692, Z -4.6667, A 0.000, B 0.000, C 0.000 }
gfCNCPoint3[21908] = {X 94.8921, Y 38.0932, Z -4.6667, A 0.000, B 0.000, C 0.000 }
gfCNCPoint3[21909] = {X 94.8910, Y 38.2309, Z -4.6667, A 0.000, B 0.000, C 0.000 }
gfCNCPoint3[21910] = {X 94.8911, Y 41.0169, Z -4.6667, A 0.000, B 0.000, C 0.000 }
gfCNCPoint3[21911] = {X 95.4382, Y 41.5559, Z -4.6667, A 0.000, B 0.000, C 0.000 }
gfCNCPoint3[21912] = {X 95.8770, Y 42.1862, Z -4.6667, A 0.000, B 0.000, C 0.000 }
gfCNCPoint3[21913] = {X 96.1089, Y 42.6639, Z -4.6667, A 0.000, B 0.000, C 0.000 }
gfCNCPoint3[21914] = {X 96.2782, Y 43.1672, Z -4.6667, A 0.000, B 0.000, C 0.000 }
gfCNCPoint3[21915] = {X 96.3813, Y 43.6833, Z -4.6667, A 0.000, B 0.000, C 0.000 }
gfCNCPoint3[21916] = {X 96.4185, Y 44.2083, Z -4.6667, A 0.000, B 0.000, C 0.000 }
gfCNCPoint3[21917] = {X 96.4184, Y 45.0392, Z -4.6667, A 0.000, B 0.000, C 0.000 }
gfCNCPoint3[21918] = {X 96.3086, Y 45.9406, Z -4.6667, A 0.000, B 0.000, C 0.000 }
gfCNCPoint3[21919] = {X 96.0023, Y 46.7954, Z -4.6667, A 0.000, B 0.000, C 0.000 }
gfCNCPoint3[21920] = {X 95.5144, Y 47.5613, Z -4.6667, A 0.000, B 0.000, C 0.000 }
gfCNCPoint3[21921] = {X 94.8692, Y 48.2003, Z -4.6667, A 0.000, B 0.000, C 0.000 }
gfCNCPoint3[21922] = {X 94.0987, Y 48.6808, Z -4.6667, A 0.000, B 0.000, C 0.000 }
gfCNCPoint3[21923] = {X 93.2410, Y 48.9789, Z -4.6667, A 0.000, B 0.000, C 0.000 }
gfCNCPoint3[21924] = {X 92.3385, Y 49.0800, Z -4.6667, A 0.000, B 0.000, C 0.000 }
gfCNCPoint3[21925] = {X 85.8951, Y 49.0800, Z -4.6667, A 0.000, B 0.000, C 0.000 }
gfCNCPoint3[21926] = {X 84.9918, Y 48.9788, Z -4.6667, A 0.000, B 0.000, C 0.000 }
gfCNCPoint3[21927] = {X 84.1334, Y 48.6801, Z -4.6667, A 0.000, B 0.000, C 0.000 }
gfCNCPoint3[21928] = {X 83.3624, Y 48.1987, Z -4.6667, A 0.000, B 0.000, C 0.000 }
gfCNCPoint3[21929] = {X 82.7171, Y 47.5586, Z -4.6667, A 0.000, B 0.000, C 0.000 }
gfCNCPoint3[21930] = {X 82.2295, Y 46.7916, Z -4.6667, A 0.000, B 0.000, C 0.000 }
gfCNCPoint3[21931] = {X 81.9238, Y 45.9356, Z -4.6667, A 0.000, B 0.000, C 0.000 }
gfCNCPoint3[21932] = {X 81.8152, Y 45.0332, Z -4.6667, A 0.000, B 0.000, C 0.000 }
gfCNCPoint3[21933] = {X 81.8151, Y 44.2084, Z -4.6667, A 0.000, B 0.000, C 0.000 }
gfCNCPoint3[21934] = {X 81.9206, Y 43.3035, Z -4.6667, A 0.000, B 0.000, C 0.000 }
gfCNCPoint3[21935] = {X 82.2216, Y 42.4435, Z -4.6667, A 0.000, B 0.000, C 0.000 }
gfCNCPoint3[21936] = {X 82.7034, Y 41.6703, Z -4.6667, A 0.000, B 0.000, C 0.000 }
gfCNCPoint3[21937] = {X 83.3428, Y 41.0213, Z -4.6667, A 0.000, B 0.000, C 0.000 }
gfCNCPoint3[21938] = {X 83.3426, Y 28.5916, Z -4.6667, A 0.000, B 0.000, C 0.000 }
gfCNCPoint3[21939] = {X 79.3426, Y 28.5916, Z -4.6667, A 0.000, B 0.000, C 0.000 }
gfCNCPoint3[21940] = {X 83.4226, Y 28.5916, Z -4.6667, A 0.000, B 0.000, C 0.000 }
gfCNCPoint3[21941] = {X 83.4225, Y 16.1223, Z -4.6667, A 0.000, B 0.000, C 0.000 }
gfCNCPoint3[21942] = {X 82.7805, Y 15.4879, Z -4.6667, A 0.000, B 0.000, C 0.000 }
gfCNCPoint3[21943] = {X 82.2971, Y 14.7258, Z -4.6667, A 0.000, B 0.000, C 0.000 }
gfCNCPoint3[21944] = {X 81.9969, Y 13.8747, Z -4.6667, A 0.000, B 0.000, C 0.000 }
gfCNCPoint3[21945] = {X 81.8951, Y 12.9779, Z -4.6667, A 0.000, B 0.000, C 0.000 }
gfCNCPoint3[21946] = {X 81.8951, Y 12.1868, Z -4.6667, A 0.000, B 0.000, C 0.000 }
gfCNCPoint3[21947] = {X 81.9954, Y 11.2967, Z -4.6667, A 0.000, B 0.000, C 0.000 }
gfCNCPoint3[21948] = {X 82.2912, Y 10.4513, Z -4.6667, A 0.000, B 0.000, C 0.000 }
gfCNCPoint3[21949] = {X 82.7677, Y 9.6929, Z -4.6667, A 0.000, B 0.000, C 0.000 }
gfCNCPoint3[21950] = {X 83.4011, Y 9.0595, Z -4.6667, A 0.000, B 0.000, C 0.000 }
gfCNCPoint3[21951] = {X 84.1595, Y 8.5829, Z -4.6667, A 0.000, B 0.000, C 0.000 }
gfCNCPoint3[21952] = {X 85.0050, Y 8.2871, Z -4.6667, A 0.000, B 0.000, C 0.000 }
gfCNCPoint3[21953] = {X 85.8951, Y 8.1868, Z -4.6667, A 0.000, B 0.000, C 0.000 }
gfCNCPoint3[21954] = {X 94.0497, Y 8.1868, Z -4.6667, A 0.000, B 0.000, C 0.000 }
gfCNCPoint3[21955] = {X 94.9398, Y 8.2871, Z -4.6667, A 0.000, B 0.000, C 0.000 }
gfCNCPoint3[21956] = {X 95.7852, Y 8.5829, Z -4.6667, A 0.000, B 0.000, C 0.000 }
gfCNCPoint3[21957] = {X 96.5436, Y 9.0595, Z -4.6667, A 0.000, B 0.000, C 0.000 }
gfCNCPoint3[21958] = {X 97.1770, Y 9.6929, Z -4.6667, A 0.000, B 0.000, C 0.000 }
gfCNCPoint3[21959] = {X 97.6535, Y 10.4513, Z -4.6667, A 0.000, B 0.000, C 0.000 }
gfCNCPoint3[21960] = {X 97.9494, Y 11.2967, Z -4.6667, A 0.000, B 0.000, C 0.000 }
gfCNCPoint3[21961] = {X 98.0497, Y 12.1868, Z -4.6667, A 0.000, B 0.000, C 0.000 }
gfCNCPoint3[21962] = {X 98.0495, Y 13.0192, Z -4.6667, A 0.000, B 0.000, C 0.000 }
gfCNCPoint3[21963] = {X 97.9794, Y 13.7245, Z -4.6667, A 0.000, B 0.000, C 0.000 }
gfCNCPoint3[21964] = {X 97.7860, Y 14.4063, Z -4.6667, A 0.000, B 0.000, C 0.000 }
gfCNCPoint3[21965] = {X 97.4752, Y 15.0434, Z -4.6667, A 0.000, B 0.000, C 0.000 }
gfCNCPoint3[21966] = {X 97.4129, Y 15.1434, Z -4.6667, A 0.000, B 0.000, C 0.000 }
gfCNCPoint3[21967] = {X 97.3476, Y 15.2415, Z -4.6667, A 0.000, B 0.000, C 0.000 }
gfCNCPoint3[21968] = {X 97.4112, Y 15.3108, Z -4.6667, A 0.000, B 0.000, C 0.000 }
gfCNCPoint3[21969] = {X 97.9968, Y 16.7687, Z -4.6667, A 0.000, B 0.000, C 0.000 }
gfCNCPoint3[21970] = {X 101.6276, Y 25.7689, Z -4.6667, A 0.000, B 0.000, C 0.000 }
gfCNCPoint3[21971] = {X 101.8768, Y 26.3795, Z -4.6667, A 0.000, B 0.000, C 0.000 }
gfCNCPoint3[21972] = {X 102.1262, Y 25.7689, Z -4.6667, A 0.000, B 0.000, C 0.000 }
gfCNCPoint3[21973] = {X 106.3419, Y 15.2553, Z -4.6667, A 0.000, B 0.000, C 0.000 }
gfCNCPoint3[21974] = {X 106.3813, Y 15.1986, Z -4.6667, A 0.000, B 0.000, C 0.000 }
gfCNCPoint3[21975] = {X 106.3234, Y 15.1094, Z -4.6667, A 0.000, B 0.000, C 0.000 }
gfCNCPoint3[21976] = {X 106.2680, Y 15.0188, Z -4.6667, A 0.000, B 0.000, C 0.000 }
gfCNCPoint3[21977] = {X 105.9604, Y 14.3756, Z -4.6667, A 0.000, B 0.000, C 0.000 }
gfCNCPoint3[21978] = {X 105.7718, Y 13.6880, Z -4.6667, A 0.000, B 0.000, C 0.000 }
gfCNCPoint3[21979] = {X 105.7083, Y 12.9779, Z -4.6667, A 0.000, B 0.000, C 0.000 }
gfCNCPoint3[21980] = {X 105.7083, Y 12.1868, Z -4.6667, A 0.000, B 0.000, C 0.000 }
gfCNCPoint3[21981] = {X 105.8086, Y 11.2967, Z -4.6667, A 0.000, B 0.000, C 0.000 }
gfCNCPoint3[21982] = {X 106.1044, Y 10.4513, Z -4.6667, A 0.000, B 0.000, C 0.000 }
gfCNCPoint3[21983] = {X 106.5810, Y 9.6929, Z -4.6667, A 0.000, B 0.000, C 0.000 }
gfCNCPoint3[21984] = {X 107.2143, Y 9.0595, Z -4.6667, A 0.000, B 0.000, C 0.000 }
gfCNCPoint3[21985] = {X 107.9727, Y 8.5829, Z -4.6667, A 0.000, B 0.000, C 0.000 }
gfCNCPoint3[21986] = {X 108.8182, Y 8.2871, Z -4.6667, A 0.000, B 0.000, C 0.000 }
gfCNCPoint3[21987] = {X 109.7083, Y 8.1868, Z -4.6667, A 0.000, B 0.000, C 0.000 }
gfCNCPoint3[21988] = {X 117.7916, Y 8.1868, Z -4.6667, A 0.000, B 0.000, C 0.000 }
gfCNCPoint3[21989] = {X 118.6817, Y 8.2871, Z -4.6667, A 0.000, B 0.000, C 0.000 }
gfCNCPoint3[21990] = {X 119.5271, Y 8.5829, Z -4.6667, A 0.000, B 0.000, C 0.000 }
gfCNCPoint3[21991] = {X 120.2855, Y 9.0595, Z -4.6667, A 0.000, B 0.000, C 0.000 }
gfCNCPoint3[21992] = {X 120.9189, Y 9.6929, Z -4.6667, A 0.000, B 0.000, C 0.000 }
gfCNCPoint3[21993] = {X 121.3955, Y 10.4513, Z -4.6667, A 0.000, B 0.000, C 0.000 }
gfCNCPoint3[21994] = {X 121.6913, Y 11.2967, Z -4.6667, A 0.000, B 0.000, C 0.000 }
gfCNCPoint3[21995] = {X 121.7916, Y 12.1868, Z -4.6667, A 0.000, B 0.000, C 0.000 }
gfCNCPoint3[21996] = {X 121.7914, Y 13.0192, Z -4.6667, A 0.000, B 0.000, C 0.000 }
gfCNCPoint3[21997] = {X 121.6828, Y 13.9045, Z -4.6667, A 0.000, B 0.000, C 0.000 }
gfCNCPoint3[21998] = {X 121.3807, Y 14.7438, Z -4.6667, A 0.000, B 0.000, C 0.000 }
gfCNCPoint3[21999] = {X 120.9002, Y 15.4952, Z -4.6667, A 0.000, B 0.000, C 0.000 }
gfCNCPoint3[22000] = {X 120.2651, Y 16.1215, Z -4.6667, A 0.000, B 0.000, C 0.000 }
gfCNCPoint3[22001] = {X 120.2640, Y 41.0659, Z -4.6667, A 0.000, B 0.000, C 0.000 }
gfCNCPoint3[22002] = {X 120.4160, Y 41.1901, Z -4.6667, A 0.000, B 0.000, C 0.000 }
gfCNCPoint3[22003] = {X 120.9967, Y 41.8157, Z -4.6667, A 0.000, B 0.000, C 0.000 }
gfCNCPoint3[22004] = {X 121.4315, Y 42.5502, Z -4.6667, A 0.000, B 0.000, C 0.000 }
gfCNCPoint3[22005] = {X 121.7005, Y 43.3602, Z -4.6667, A 0.000, B 0.000, C 0.000 }
gfCNCPoint3[22006] = {X 121.7916, Y 44.2089, Z -4.6667, A 0.000, B 0.000, C 0.000 }
gfCNCPoint3[22007] = {X 121.7916, Y 45.0000, Z -4.6667, A 0.000, B 0.000, C 0.000 }
gfCNCPoint3[22008] = {X 121.6913, Y 45.8901, Z -4.6667, A 0.000, B 0.000, C 0.000 }
gfCNCPoint3[22009] = {X 121.3955, Y 46.7355, Z -4.6667, A 0.000, B 0.000, C 0.000 }
gfCNCPoint3[22010] = {X 120.9189, Y 47.4940, Z -4.6667, A 0.000, B 0.000, C 0.000 }
gfCNCPoint3[22011] = {X 120.2855, Y 48.1273, Z -4.6667, A 0.000, B 0.000, C 0.000 }
gfCNCPoint3[22012] = {X 119.5271, Y 48.6039, Z -4.6667, A 0.000, B 0.000, C 0.000 }
gfCNCPoint3[22013] = {X 118.6817, Y 48.8997, Z -4.6667, A 0.000, B 0.000, C 0.000 }
gfCNCPoint3[22014] = {X 117.7916, Y 49.0000, Z -4.6667, A 0.000, B 0.000, C 0.000 }
gfCNCPoint3[22015] = {X 111.9185, Y 49.0000, Z -4.6667, A 0.000, B 0.000, C 0.000 }
gfCNCPoint3[22016] = {X 111.0284, Y 48.8997, Z -4.6667, A 0.000, B 0.000, C 0.000 }
gfCNCPoint3[22017] = {X 110.1829, Y 48.6039, Z -4.6667, A 0.000, B 0.000, C 0.000 }
gfCNCPoint3[22018] = {X 109.4245, Y 48.1273, Z -4.6667, A 0.000, B 0.000, C 0.000 }
gfCNCPoint3[22019] = {X 108.7911, Y 47.4939, Z -4.6667, A 0.000, B 0.000, C 0.000 }
gfCNCPoint3[22020] = {X 108.3146, Y 46.7355, Z -4.6667, A 0.000, B 0.000, C 0.000 }
gfCNCPoint3[22021] = {X 108.0188, Y 45.8901, Z -4.6667, A 0.000, B 0.000, C 0.000 }
gfCNCPoint3[22022] = {X 107.9185, Y 45.0000, Z -4.6667, A 0.000, B 0.000, C 0.000 }
gfCNCPoint3[22023] = {X 107.9185, Y 44.1775, Z -4.6667, A 0.000, B 0.000, C 0.000 }
gfCNCPoint3[22024] = {X 107.9512, Y 43.6779, Z -4.6667, A 0.000, B 0.000, C 0.000 }
gfCNCPoint3[22025] = {X 108.0489, Y 43.1868, Z -4.6667, A 0.000, B 0.000, C 0.000 }
gfCNCPoint3[22026] = {X 108.2036, Y 42.7278, Z -4.6667, A 0.000, B 0.000, C 0.000 }
gfCNCPoint3[22027] = {X 108.4150, Y 42.2921, Z -4.6667, A 0.000, B 0.000, C 0.000 }
gfCNCPoint3[22028] = {X 108.4387, Y 42.2509, Z -4.6667, A 0.000, B 0.000, C 0.000 }
gfCNCPoint3[22029] = {X 108.4629, Y 42.2099, Z -4.6667, A 0.000, B 0.000, C 0.000 }
gfCNCPoint3[22030] = {X 108.9113, Y 41.5698, Z -4.6667, A 0.000, B 0.000, C 0.000 }
gfCNCPoint3[22031] = {X 109.4459, Y 40.9999, Z -4.6667, A 0.000, B 0.000, C 0.000 }
gfCNCPoint3[22032] = {X 109.4458, Y 38.9229, Z -4.6667, A 0.000, B 0.000, C 0.000 }
gfCNCPoint3[22033] = {X 108.9328, Y 38.9229, Z -4.6667, A 0.000, B 0.000, C 0.000 }
gfCNCPoint3[22034] = {X 105.8164, Y 46.5384, Z -4.6667, A 0.000, B 0.000, C 0.000 }
gfCNCPoint3[22035] = {X 105.3339, Y 47.3869, Z -4.6667, A 0.000, B 0.000, C 0.000 }
gfCNCPoint3[22036] = {X 104.6602, Y 48.0932, Z -4.6667, A 0.000, B 0.000, C 0.000 }
gfCNCPoint3[22037] = {X 103.8355, Y 48.6154, Z -4.6667, A 0.000, B 0.000, C 0.000 }
gfCNCPoint3[22038] = {X 102.9580, Y 48.9121, Z -4.6667, A 0.000, B 0.000, C 0.000 }
gfCNCPoint3[22039] = {X 102.0357, Y 48.9990, Z -4.6667, A 0.000, B 0.000, C 0.000 }
gfCNCPoint3[22040] = {X 101.1182, Y 48.8715, Z -4.6667, A 0.000, B 0.000, C 0.000 }
gfCNCPoint3[22041] = {X 100.2546, Y 48.5362, Z -4.6667, A 0.000, B 0.000, C 0.000 }
gfCNCPoint3[22042] = {X 99.4912, Y 48.0114, Z -4.6667, A 0.000, B 0.000, C 0.000 }
gfCNCPoint3[22043] = {X 98.8691, Y 47.3250, Z -4.6667, A 0.000, B 0.000, C 0.000 }
gfCNCPoint3[22044] = {X 98.4216, Y 46.5139, Z -4.6667, A 0.000, B 0.000, C 0.000 }
gfCNCPoint3[22045] = {X 94.8152, Y 37.6939, Z -4.6667, A 0.000, B 0.000, C 0.000 }
gfCNCPoint3[22046] = {X 94.8110, Y 38.2306, Z -4.6667, A 0.000, B 0.000, C 0.000 }
gfCNCPoint3[22047] = {X 94.8111, Y 41.0550, Z -4.6667, A 0.000, B 0.000, C 0.000 }
gfCNCPoint3[22048] = {X 95.3649, Y 41.5930, Z -4.6667, A 0.000, B 0.000, C 0.000 }
gfCNCPoint3[22049] = {X 95.8074, Y 42.2257, Z -4.6667, A 0.000, B 0.000, C 0.000 }
gfCNCPoint3[22050] = {X 96.0349, Y 42.6942, Z -4.6667, A 0.000, B 0.000, C 0.000 }
gfCNCPoint3[22051] = {X 96.2009, Y 43.1879, Z -4.6667, A 0.000, B 0.000, C 0.000 }
gfCNCPoint3[22052] = {X 96.3020, Y 43.6940, Z -4.6667, A 0.000, B 0.000, C 0.000 }
gfCNCPoint3[22053] = {X 96.3385, Y 44.2089, Z -4.6667, A 0.000, B 0.000, C 0.000 }
gfCNCPoint3[22054] = {X 96.3384, Y 45.0384, Z -4.6667, A 0.000, B 0.000, C 0.000 }
gfCNCPoint3[22055] = {X 96.2308, Y 45.9222, Z -4.6667, A 0.000, B 0.000, C 0.000 }
gfCNCPoint3[22056] = {X 95.9304, Y 46.7602, Z -4.6667, A 0.000, B 0.000, C 0.000 }
gfCNCPoint3[22057] = {X 95.4521, Y 47.5111, Z -4.6667, A 0.000, B 0.000, C 0.000 }
gfCNCPoint3[22058] = {X 94.8196, Y 48.1376, Z -4.6667, A 0.000, B 0.000, C 0.000 }
gfCNCPoint3[22059] = {X 94.0642, Y 48.6086, Z -4.6667, A 0.000, B 0.000, C 0.000 }
gfCNCPoint3[22060] = {X 93.2233, Y 48.9009, Z -4.6667, A 0.000, B 0.000, C 0.000 }
gfCNCPoint3[22061] = {X 92.3385, Y 49.0000, Z -4.6667, A 0.000, B 0.000, C 0.000 }
gfCNCPoint3[22062] = {X 85.8951, Y 49.0000, Z -4.6667, A 0.000, B 0.000, C 0.000 }
gfCNCPoint3[22063] = {X 85.0050, Y 48.8997, Z -4.6667, A 0.000, B 0.000, C 0.000 }
gfCNCPoint3[22064] = {X 84.1595, Y 48.6039, Z -4.6667, A 0.000, B 0.000, C 0.000 }
gfCNCPoint3[22065] = {X 83.4011, Y 48.1273, Z -4.6667, A 0.000, B 0.000, C 0.000 }
gfCNCPoint3[22066] = {X 82.7677, Y 47.4939, Z -4.6667, A 0.000, B 0.000, C 0.000 }
gfCNCPoint3[22067] = {X 82.2912, Y 46.7355, Z -4.6667, A 0.000, B 0.000, C 0.000 }
gfCNCPoint3[22068] = {X 81.9954, Y 45.8901, Z -4.6667, A 0.000, B 0.000, C 0.000 }
gfCNCPoint3[22069] = {X 81.8951, Y 45.0000, Z -4.6667, A 0.000, B 0.000, C 0.000 }
gfCNCPoint3[22070] = {X 81.8951, Y 44.2089, Z -4.6667, A 0.000, B 0.000, C 0.000 }
gfCNCPoint3[22071] = {X 82.0007, Y 43.3122, Z -4.6667, A 0.000, B 0.000, C 0.000 }
gfCNCPoint3[22072] = {X 82.3019, Y 42.4610, Z -4.6667, A 0.000, B 0.000, C 0.000 }
gfCNCPoint3[22073] = {X 82.7839, Y 41.6976, Z -4.6667, A 0.000, B 0.000, C 0.000 }
gfCNCPoint3[22074] = {X 83.4228, Y 41.0596, Z -4.6667, A 0.000, B 0.000, C 0.000 }
gfCNCPoint3[22075] = {X 83.4226, Y 28.5916, Z -4.6667, A 0.000, B 0.000, C 0.000 }
gfCNCPoint3[22076] = {X 79.3426, Y 28.5916, Z -4.6667, A 0.000, B 0.000, C 0.000 }
gfCNCPoint3[22077] = {X 79.3426, Y 28.5916, Z -1.6667, A 0.000, B 0.000, C 0.000 }
gfCNCPoint3[22078] = {X 79.3426, Y 28.5916, Z 11.0000, A 0.000, B 0.000, C 0.000 }
gfCNCPoint3[22079] = {X 136.1636, Y 30.3966, Z 11.0000, A 0.000, B 0.000, C 0.000 }
gfCNCPoint3[22080] = {X 136.1636, Y 30.3966, Z -1.6667, A 0.000, B 0.000, C 0.000 }
gfCNCPoint3[22081] = {X 136.1636, Y 30.3966, Z -4.6667, A 0.000, B 0.000, C 0.000 }
gfCNCPoint3[22082] = {X 140.2436, Y 30.3966, Z -4.6667, A 0.000, B 0.000, C 0.000 }
gfCNCPoint3[22083] = {X 140.2436, Y 19.8775, Z -4.6667, A 0.000, B 0.000, C 0.000 }
gfCNCPoint3[22084] = {X 137.4240, Y 19.8769, Z -4.6667, A 0.000, B 0.000, C 0.000 }
gfCNCPoint3[22085] = {X 136.8916, Y 20.5216, Z -4.6667, A 0.000, B 0.000, C 0.000 }
gfCNCPoint3[22086] = {X 136.2450, Y 21.0517, Z -4.6667, A 0.000, B 0.000, C 0.000 }
gfCNCPoint3[22087] = {X 135.5084, Y 21.4473, Z -4.6667, A 0.000, B 0.000, C 0.000 }
gfCNCPoint3[22088] = {X 134.7093, Y 21.6936, Z -4.6667, A 0.000, B 0.000, C 0.000 }
gfCNCPoint3[22089] = {X 133.8778, Y 21.7814, Z -4.6667, A 0.000, B 0.000, C 0.000 }
gfCNCPoint3[22090] = {X 133.2006, Y 21.7815, Z -4.6667, A 0.000, B 0.000, C 0.000 }
gfCNCPoint3[22091] = {X 132.2394, Y 21.6732, Z -4.6667, A 0.000, B 0.000, C 0.000 }
gfCNCPoint3[22092] = {X 131.3263, Y 21.3537, Z -4.6667, A 0.000, B 0.000, C 0.000 }
gfCNCPoint3[22093] = {X 130.5072, Y 20.8390, Z -4.6667, A 0.000, B 0.000, C 0.000 }
gfCNCPoint3[22094] = {X 129.8231, Y 20.1550, Z -4.6667, A 0.000, B 0.000, C 0.000 }
gfCNCPoint3[22095] = {X 129.3085, Y 19.3359, Z -4.6667, A 0.000, B 0.000, C 0.000 }
gfCNCPoint3[22096] = {X 128.9890, Y 18.4228, Z -4.6667, A 0.000, B 0.000, C 0.000 }
gfCNCPoint3[22097] = {X 128.8806, Y 17.4615, Z -4.6667, A 0.000, B 0.000, C 0.000 }
gfCNCPoint3[22098] = {X 128.8806, Y 10.4835, Z -4.6667, A 0.000, B 0.000, C 0.000 }
gfCNCPoint3[22099] = {X 128.9874, Y 9.5289, Z -4.6667, A 0.000, B 0.000, C 0.000 }
gfCNCPoint3[22100] = {X 129.3026, Y 8.6214, Z -4.6667, A 0.000, B 0.000, C 0.000 }
gfCNCPoint3[22101] = {X 129.8104, Y 7.8061, Z -4.6667, A 0.000, B 0.000, C 0.000 }
gfCNCPoint3[22102] = {X 130.4859, Y 7.1231, Z -4.6667, A 0.000, B 0.000, C 0.000 }
gfCNCPoint3[22103] = {X 131.2956, Y 6.6063, Z -4.6667, A 0.000, B 0.000, C 0.000 }
gfCNCPoint3[22104] = {X 132.1995, Y 6.2811, Z -4.6667, A 0.000, B 0.000, C 0.000 }
gfCNCPoint3[22105] = {X 133.1529, Y 6.1638, Z -4.6667, A 0.000, B 0.000, C 0.000 }
gfCNCPoint3[22106] = {X 133.8866, Y 6.1637, Z -4.6667, A 0.000, B 0.000, C 0.000 }
gfCNCPoint3[22107] = {X 134.7111, Y 6.2518, Z -4.6667, A 0.000, B 0.000, C 0.000 }
gfCNCPoint3[22108] = {X 135.5035, Y 6.4957, Z -4.6667, A 0.000, B 0.000, C 0.000 }
gfCNCPoint3[22109] = {X 136.2348, Y 6.8865, Z -4.6667, A 0.000, B 0.000, C 0.000 }
gfCNCPoint3[22110] = {X 136.8779, Y 7.4098, Z -4.6667, A 0.000, B 0.000, C 0.000 }
gfCNCPoint3[22111] = {X 137.4092, Y 8.0464, Z -4.6667, A 0.000, B 0.000, C 0.000 }
gfCNCPoint3[22112] = {X 155.1127, Y 8.0476, Z -4.6667, A 0.000, B 0.000, C 0.000 }
gfCNCPoint3[22113] = {X 155.6447, Y 7.4099, Z -4.6667, A 0.000, B 0.000, C 0.000 }
gfCNCPoint3[22114] = {X 156.2889, Y 6.8859, Z -4.6667, A 0.000, B 0.000, C 0.000 }
gfCNCPoint3[22115] = {X 157.0215, Y 6.4947, Z -4.6667, A 0.000, B 0.000, C 0.000 }
gfCNCPoint3[22116] = {X 157.8154, Y 6.2510, Z -4.6667, A 0.000, B 0.000, C 0.000 }
gfCNCPoint3[22117] = {X 158.6412, Y 6.1637, Z -4.6667, A 0.000, B 0.000, C 0.000 }
gfCNCPoint3[22118] = {X 159.3781, Y 6.1639, Z -4.6667, A 0.000, B 0.000, C 0.000 }
gfCNCPoint3[22119] = {X 160.3301, Y 6.2828, Z -4.6667, A 0.000, B 0.000, C 0.000 }
gfCNCPoint3[22120] = {X 161.2324, Y 6.6088, Z -4.6667, A 0.000, B 0.000, C 0.000 }
gfCNCPoint3[22121] = {X 162.0405, Y 7.1260, Z -4.6667, A 0.000, B 0.000, C 0.000 }
gfCNCPoint3[22122] = {X 162.7145, Y 7.8088, Z -4.6667, A 0.000, B 0.000, C 0.000 }
gfCNCPoint3[22123] = {X 163.2212, Y 8.6236, Z -4.6667, A 0.000, B 0.000, C 0.000 }
gfCNCPoint3[22124] = {X 163.5355, Y 9.5300, Z -4.6667, A 0.000, B 0.000, C 0.000 }
gfCNCPoint3[22125] = {X 163.6421, Y 10.4835, Z -4.6667, A 0.000, B 0.000, C 0.000 }
gfCNCPoint3[22126] = {X 163.6421, Y 17.4615, Z -4.6667, A 0.000, B 0.000, C 0.000 }
gfCNCPoint3[22127] = {X 163.5355, Y 18.4152, Z -4.6667, A 0.000, B 0.000, C 0.000 }
gfCNCPoint3[22128] = {X 163.2211, Y 19.3218, Z -4.6667, A 0.000, B 0.000, C 0.000 }
gfCNCPoint3[22129] = {X 162.7142, Y 20.1366, Z -4.6667, A 0.000, B 0.000, C 0.000 }
gfCNCPoint3[22130] = {X 162.0400, Y 20.8194, Z -4.6667, A 0.000, B 0.000, C 0.000 }
gfCNCPoint3[22131] = {X 161.2318, Y 21.3365, Z -4.6667, A 0.000, B 0.000, C 0.000 }
gfCNCPoint3[22132] = {X 160.3292, Y 21.6625, Z -4.6667, A 0.000, B 0.000, C 0.000 }
gfCNCPoint3[22133] = {X 159.3770, Y 21.7812, Z -4.6667, A 0.000, B 0.000, C 0.000 }
gfCNCPoint3[22134] = {X 158.6792, Y 21.7815, Z -4.6667, A 0.000, B 0.000, C 0.000 }
gfCNCPoint3[22135] = {X 157.8408, Y 21.6965, Z -4.6667, A 0.000, B 0.000, C 0.000 }
gfCNCPoint3[22136] = {X 157.0346, Y 21.4516, Z -4.6667, A 0.000, B 0.000, C 0.000 }
gfCNCPoint3[22137] = {X 156.2906, Y 21.0560, Z -4.6667, A 0.000, B 0.000, C 0.000 }
gfCNCPoint3[22138] = {X 155.6367, Y 20.5244, Z -4.6667, A 0.000, B 0.000, C 0.000 }
gfCNCPoint3[22139] = {X 155.0974, Y 19.8769, Z -4.6667, A 0.000, B 0.000, C 0.000 }
gfCNCPoint3[22140] = {X 152.2765, Y 19.8781, Z -4.6667, A 0.000, B 0.000, C 0.000 }
gfCNCPoint3[22141] = {X 152.2751, Y 40.8742, Z -4.6667, A 0.000, B 0.000, C 0.000 }
gfCNCPoint3[22142] = {X 152.7409, Y 41.3756, Z -4.6667, A 0.000, B 0.000, C 0.000 }
gfCNCPoint3[22143] = {X 152.8358, Y 41.4888, Z -4.6667, A 0.000, B 0.000, C 0.000 }
gfCNCPoint3[22144] = {X 153.3614, Y 42.3141, Z -4.6667, A 0.000, B 0.000, C 0.000 }
gfCNCPoint3[22145] = {X 153.6893, Y 43.2359, Z -4.6667, A 0.000, B 0.000, C 0.000 }
gfCNCPoint3[22146] = {X 153.8031, Y 44.2076, Z -4.6667, A 0.000, B 0.000, C 0.000 }
gfCNCPoint3[22147] = {X 153.8029, Y 45.0415, Z -4.6667, A 0.000, B 0.000, C 0.000 }
gfCNCPoint3[22148] = {X 153.6867, Y 45.9960, Z -4.6667, A 0.000, B 0.000, C 0.000 }
gfCNCPoint3[22149] = {X 153.3623, Y 46.9011, Z -4.6667, A 0.000, B 0.000, C 0.000 }
gfCNCPoint3[22150] = {X 152.8458, Y 47.7120, Z -4.6667, A 0.000, B 0.000, C 0.000 }
gfCNCPoint3[22151] = {X 152.1626, Y 48.3886, Z -4.6667, A 0.000, B 0.000, C 0.000 }
gfCNCPoint3[22152] = {X 151.3468, Y 48.8973, Z -4.6667, A 0.000, B 0.000, C 0.000 }
gfCNCPoint3[22153] = {X 150.4386, Y 49.2130, Z -4.6667, A 0.000, B 0.000, C 0.000 }
gfCNCPoint3[22154] = {X 149.4831, Y 49.3200, Z -4.6667, A 0.000, B 0.000, C 0.000 }
gfCNCPoint3[22155] = {X 143.0396, Y 49.3200, Z -4.6667, A 0.000, B 0.000, C 0.000 }
gfCNCPoint3[22156] = {X 142.0831, Y 49.2128, Z -4.6667, A 0.000, B 0.000, C 0.000 }
gfCNCPoint3[22157] = {X 141.1741, Y 48.8964, Z -4.6667, A 0.000, B 0.000, C 0.000 }
gfCNCPoint3[22158] = {X 140.3576, Y 48.3866, Z -4.6667, A 0.000, B 0.000, C 0.000 }
gfCNCPoint3[22159] = {X 139.6743, Y 47.7087, Z -4.6667, A 0.000, B 0.000, C 0.000 }
gfCNCPoint3[22160] = {X 139.1581, Y 46.8964, Z -4.6667, A 0.000, B 0.000, C 0.000 }
gfCNCPoint3[22161] = {X 138.8346, Y 45.9899, Z -4.6667, A 0.000, B 0.000, C 0.000 }
gfCNCPoint3[22162] = {X 138.7198, Y 45.0342, Z -4.6667, A 0.000, B 0.000, C 0.000 }
gfCNCPoint3[22163] = {X 138.7200, Y 44.1494, Z -4.6667, A 0.000, B 0.000, C 0.000 }
gfCNCPoint3[22164] = {X 138.8305, Y 43.2364, Z -4.6667, A 0.000, B 0.000, C 0.000 }
gfCNCPoint3[22165] = {X 139.1317, Y 42.3675, Z -4.6667, A 0.000, B 0.000, C 0.000 }
gfCNCPoint3[22166] = {X 139.6099, Y 41.5821, Z -4.6667, A 0.000, B 0.000, C 0.000 }
gfCNCPoint3[22167] = {X 140.2436, Y 40.9157, Z -4.6667, A 0.000, B 0.000, C 0.000 }
gfCNCPoint3[22168] = {X 140.2436, Y 30.3966, Z -4.6667, A 0.000, B 0.000, C 0.000 }
gfCNCPoint3[22169] = {X 136.2436, Y 30.3966, Z -4.6667, A 0.000, B 0.000, C 0.000 }
gfCNCPoint3[22170] = {X 140.3236, Y 30.3966, Z -4.6667, A 0.000, B 0.000, C 0.000 }
gfCNCPoint3[22171] = {X 140.3236, Y 19.7975, Z -4.6667, A 0.000, B 0.000, C 0.000 }
gfCNCPoint3[22172] = {X 137.3796, Y 19.7969, Z -4.6667, A 0.000, B 0.000, C 0.000 }
gfCNCPoint3[22173] = {X 137.3568, Y 19.8335, Z -4.6667, A 0.000, B 0.000, C 0.000 }
gfCNCPoint3[22174] = {X 136.8342, Y 20.4659, Z -4.6667, A 0.000, B 0.000, C 0.000 }
gfCNCPoint3[22175] = {X 136.1997, Y 20.9858, Z -4.6667, A 0.000, B 0.000, C 0.000 }
gfCNCPoint3[22176] = {X 135.4769, Y 21.3738, Z -4.6667, A 0.000, B 0.000, C 0.000 }
gfCNCPoint3[22177] = {X 134.6930, Y 21.6153, Z -4.6667, A 0.000, B 0.000, C 0.000 }
gfCNCPoint3[22178] = {X 133.8772, Y 21.7014, Z -4.6667, A 0.000, B 0.000, C 0.000 }
gfCNCPoint3[22179] = {X 133.2006, Y 21.7015, Z -4.6667, A 0.000, B 0.000, C 0.000 }
gfCNCPoint3[22180] = {X 132.2572, Y 21.5952, Z -4.6667, A 0.000, B 0.000, C 0.000 }
gfCNCPoint3[22181] = {X 131.3610, Y 21.2816, Z -4.6667, A 0.000, B 0.000, C 0.000 }
gfCNCPoint3[22182] = {X 130.5570, Y 20.7765, Z -4.6667, A 0.000, B 0.000, C 0.000 }
gfCNCPoint3[22183] = {X 129.8857, Y 20.1051, Z -4.6667, A 0.000, B 0.000, C 0.000 }
gfCNCPoint3[22184] = {X 129.3805, Y 19.3012, Z -4.6667, A 0.000, B 0.000, C 0.000 }
gfCNCPoint3[22185] = {X 129.0669, Y 18.4050, Z -4.6667, A 0.000, B 0.000, C 0.000 }
gfCNCPoint3[22186] = {X 128.9606, Y 17.4615, Z -4.6667, A 0.000, B 0.000, C 0.000 }
gfCNCPoint3[22187] = {X 128.9606, Y 10.4835, Z -4.6667, A 0.000, B 0.000, C 0.000 }
gfCNCPoint3[22188] = {X 129.0655, Y 9.5466, Z -4.6667, A 0.000, B 0.000, C 0.000 }
gfCNCPoint3[22189] = {X 129.3747, Y 8.6559, Z -4.6667, A 0.000, B 0.000, C 0.000 }
gfCNCPoint3[22190] = {X 129.8732, Y 7.8557, Z -4.6667, A 0.000, B 0.000, C 0.000 }
gfCNCPoint3[22191] = {X 130.5362, Y 7.1853, Z -4.6667, A 0.000, B 0.000, C 0.000 }
gfCNCPoint3[22192] = {X 131.3309, Y 6.6781, Z -4.6667, A 0.000, B 0.000, C 0.000 }
gfCNCPoint3[22193] = {X 132.2180, Y 6.3589, Z -4.6667, A 0.000, B 0.000, C 0.000 }
gfCNCPoint3[22194] = {X 133.1538, Y 6.2438, Z -4.6667, A 0.000, B 0.000, C 0.000 }
gfCNCPoint3[22195] = {X 133.8858, Y 6.2437, Z -4.6667, A 0.000, B 0.000, C 0.000 }
gfCNCPoint3[22196] = {X 134.7032, Y 6.3318, Z -4.6667, A 0.000, B 0.000, C 0.000 }
gfCNCPoint3[22197] = {X 135.4883, Y 6.5760, Z -4.6667, A 0.000, B 0.000, C 0.000 }
gfCNCPoint3[22198] = {X 136.2114, Y 6.9672, Z -4.6667, A 0.000, B 0.000, C 0.000 }
gfCNCPoint3[22199] = {X 136.8455, Y 7.4905, Z -4.6667, A 0.000, B 0.000, C 0.000 }
gfCNCPoint3[22200] = {X 137.3667, Y 8.1264, Z -4.6667, A 0.000, B 0.000, C 0.000 }
gfCNCPoint3[22201] = {X 155.1552, Y 8.1276, Z -4.6667, A 0.000, B 0.000, C 0.000 }
gfCNCPoint3[22202] = {X 155.6771, Y 7.4906, Z -4.6667, A 0.000, B 0.000, C 0.000 }
gfCNCPoint3[22203] = {X 156.3122, Y 6.9665, Z -4.6667, A 0.000, B 0.000, C 0.000 }
gfCNCPoint3[22204] = {X 157.0367, Y 6.5751, Z -4.6667, A 0.000, B 0.000, C 0.000 }
gfCNCPoint3[22205] = {X 157.8231, Y 6.3311, Z -4.6667, A 0.000, B 0.000, C 0.000 }
gfCNCPoint3[22206] = {X 158.6420, Y 6.2437, Z -4.6667, A 0.000, B 0.000, C 0.000 }
gfCNCPoint3[22207] = {X 159.3770, Y 6.2439, Z -4.6667, A 0.000, B 0.000, C 0.000 }
gfCNCPoint3[22208] = {X 160.3114, Y 6.3606, Z -4.6667, A 0.000, B 0.000, C 0.000 }
gfCNCPoint3[22209] = {X 161.1970, Y 6.6806, Z -4.6667, A 0.000, B 0.000, C 0.000 }
gfCNCPoint3[22210] = {X 161.9902, Y 7.1882, Z -4.6667, A 0.000, B 0.000, C 0.000 }
gfCNCPoint3[22211] = {X 162.6517, Y 7.8584, Z -4.6667, A 0.000, B 0.000, C 0.000 }
gfCNCPoint3[22212] = {X 163.1490, Y 8.6580, Z -4.6667, A 0.000, B 0.000, C 0.000 }
gfCNCPoint3[22213] = {X 163.4575, Y 9.5477, Z -4.6667, A 0.000, B 0.000, C 0.000 }
gfCNCPoint3[22214] = {X 163.5621, Y 10.4835, Z -4.6667, A 0.000, B 0.000, C 0.000 }
gfCNCPoint3[22215] = {X 163.5621, Y 17.4615, Z -4.6667, A 0.000, B 0.000, C 0.000 }
gfCNCPoint3[22216] = {X 163.4575, Y 18.3975, Z -4.6667, A 0.000, B 0.000, C 0.000 }
gfCNCPoint3[22217] = {X 163.1489, Y 19.2873, Z -4.6667, A 0.000, B 0.000, C 0.000 }
gfCNCPoint3[22218] = {X 162.6514, Y 20.0870, Z -4.6667, A 0.000, B 0.000, C 0.000 }
gfCNCPoint3[22219] = {X 161.9897, Y 20.7572, Z -4.6667, A 0.000, B 0.000, C 0.000 }
gfCNCPoint3[22220] = {X 161.1964, Y 21.2648, Z -4.6667, A 0.000, B 0.000, C 0.000 }
gfCNCPoint3[22221] = {X 160.3106, Y 21.5847, Z -4.6667, A 0.000, B 0.000, C 0.000 }
gfCNCPoint3[22222] = {X 159.3760, Y 21.7012, Z -4.6667, A 0.000, B 0.000, C 0.000 }
gfCNCPoint3[22223] = {X 158.6795, Y 21.7015, Z -4.6667, A 0.000, B 0.000, C 0.000 }
gfCNCPoint3[22224] = {X 157.8483, Y 21.6164, Z -4.6667, A 0.000, B 0.000, C 0.000 }
gfCNCPoint3[22225] = {X 157.0495, Y 21.3712, Z -4.6667, A 0.000, B 0.000, C 0.000 }
gfCNCPoint3[22226] = {X 156.3137, Y 20.9752, Z -4.6667, A 0.000, B 0.000, C 0.000 }
gfCNCPoint3[22227] = {X 155.6690, Y 20.4437, Z -4.6667, A 0.000, B 0.000, C 0.000 }
gfCNCPoint3[22228] = {X 155.1400, Y 19.7969, Z -4.6667, A 0.000, B 0.000, C 0.000 }
gfCNCPoint3[22229] = {X 152.1965, Y 19.7981, Z -4.6667, A 0.000, B 0.000, C 0.000 }
gfCNCPoint3[22230] = {X 152.1951, Y 40.9056, Z -4.6667, A 0.000, B 0.000, C 0.000 }
gfCNCPoint3[22231] = {X 152.6809, Y 41.4286, Z -4.6667, A 0.000, B 0.000, C 0.000 }
gfCNCPoint3[22232] = {X 152.7741, Y 41.5397, Z -4.6667, A 0.000, B 0.000, C 0.000 }
gfCNCPoint3[22233] = {X 153.2897, Y 42.3496, Z -4.6667, A 0.000, B 0.000, C 0.000 }
gfCNCPoint3[22234] = {X 153.6114, Y 43.2543, Z -4.6667, A 0.000, B 0.000, C 0.000 }
gfCNCPoint3[22235] = {X 153.7231, Y 44.2079, Z -4.6667, A 0.000, B 0.000, C 0.000 }
gfCNCPoint3[22236] = {X 153.7229, Y 45.0408, Z -4.6667, A 0.000, B 0.000, C 0.000 }
gfCNCPoint3[22237] = {X 153.6089, Y 45.9775, Z -4.6667, A 0.000, B 0.000, C 0.000 }
gfCNCPoint3[22238] = {X 153.2905, Y 46.8659, Z -4.6667, A 0.000, B 0.000, C 0.000 }
gfCNCPoint3[22239] = {X 152.7835, Y 47.6618, Z -4.6667, A 0.000, B 0.000, C 0.000 }
gfCNCPoint3[22240] = {X 152.1130, Y 48.3258, Z -4.6667, A 0.000, B 0.000, C 0.000 }
gfCNCPoint3[22241] = {X 151.3123, Y 48.8251, Z -4.6667, A 0.000, B 0.000, C 0.000 }
gfCNCPoint3[22242] = {X 150.4209, Y 49.1350, Z -4.6667, A 0.000, B 0.000, C 0.000 }
gfCNCPoint3[22243] = {X 149.4831, Y 49.2400, Z -4.6667, A 0.000, B 0.000, C 0.000 }
gfCNCPoint3[22244] = {X 143.0396, Y 49.2400, Z -4.6667, A 0.000, B 0.000, C 0.000 }
gfCNCPoint3[22245] = {X 142.1008, Y 49.1348, Z -4.6667, A 0.000, B 0.000, C 0.000 }
gfCNCPoint3[22246] = {X 141.2086, Y 48.8243, Z -4.6667, A 0.000, B 0.000, C 0.000 }
gfCNCPoint3[22247] = {X 140.4073, Y 48.3239, Z -4.6667, A 0.000, B 0.000, C 0.000 }
gfCNCPoint3[22248] = {X 139.7367, Y 47.6586, Z -4.6667, A 0.000, B 0.000, C 0.000 }
gfCNCPoint3[22249] = {X 139.2300, Y 46.8612, Z -4.6667, A 0.000, B 0.000, C 0.000 }
gfCNCPoint3[22250] = {X 138.9124, Y 45.9715, Z -4.6667, A 0.000, B 0.000, C 0.000 }
gfCNCPoint3[22251] = {X 138.7998, Y 45.0336, Z -4.6667, A 0.000, B 0.000, C 0.000 }
gfCNCPoint3[22252] = {X 138.8000, Y 44.1505, Z -4.6667, A 0.000, B 0.000, C 0.000 }
gfCNCPoint3[22253] = {X 138.9105, Y 43.2454, Z -4.6667, A 0.000, B 0.000, C 0.000 }
gfCNCPoint3[22254] = {X 139.2119, Y 42.3850, Z -4.6667, A 0.000, B 0.000, C 0.000 }
gfCNCPoint3[22255] = {X 139.6903, Y 41.6088, Z -4.6667, A 0.000, B 0.000, C 0.000 }
gfCNCPoint3[22256] = {X 140.3236, Y 40.9529, Z -4.6667, A 0.000, B 0.000, C 0.000 }
gfCNCPoint3[22257] = {X 140.3236, Y 30.3966, Z -4.6667, A 0.000, B 0.000, C 0.000 }
gfCNCPoint3[22258] = {X 136.3236, Y 30.3966, Z -4.6667, A 0.000, B 0.000, C 0.000 }
gfCNCPoint3[22259] = {X 140.4036, Y 30.3966, Z -4.6667, A 0.000, B 0.000, C 0.000 }
gfCNCPoint3[22260] = {X 140.4036, Y 19.7175, Z -4.6667, A 0.000, B 0.000, C 0.000 }
gfCNCPoint3[22261] = {X 137.3353, Y 19.7169, Z -4.6667, A 0.000, B 0.000, C 0.000 }
gfCNCPoint3[22262] = {X 137.2897, Y 19.7899, Z -4.6667, A 0.000, B 0.000, C 0.000 }
gfCNCPoint3[22263] = {X 136.7770, Y 20.4100, Z -4.6667, A 0.000, B 0.000, C 0.000 }
gfCNCPoint3[22264] = {X 136.1545, Y 20.9198, Z -4.6667, A 0.000, B 0.000, C 0.000 }
gfCNCPoint3[22265] = {X 135.4456, Y 21.3002, Z -4.6667, A 0.000, B 0.000, C 0.000 }
gfCNCPoint3[22266] = {X 134.6766, Y 21.5370, Z -4.6667, A 0.000, B 0.000, C 0.000 }
gfCNCPoint3[22267] = {X 133.8765, Y 21.6214, Z -4.6667, A 0.000, B 0.000, C 0.000 }
gfCNCPoint3[22268] = {X 133.2006, Y 21.6215, Z -4.6667, A 0.000, B 0.000, C 0.000 }
gfCNCPoint3[22269] = {X 132.2750, Y 21.5172, Z -4.6667, A 0.000, B 0.000, C 0.000 }
gfCNCPoint3[22270] = {X 131.3957, Y 21.2096, Z -4.6667, A 0.000, B 0.000, C 0.000 }
gfCNCPoint3[22271] = {X 130.6069, Y 20.7140, Z -4.6667, A 0.000, B 0.000, C 0.000 }
gfCNCPoint3[22272] = {X 129.9482, Y 20.0553, Z -4.6667, A 0.000, B 0.000, C 0.000 }
gfCNCPoint3[22273] = {X 129.4526, Y 19.2665, Z -4.6667, A 0.000, B 0.000, C 0.000 }
gfCNCPoint3[22274] = {X 129.1449, Y 18.3872, Z -4.6667, A 0.000, B 0.000, C 0.000 }
gfCNCPoint3[22275] = {X 129.0406, Y 17.4615, Z -4.6667, A 0.000, B 0.000, C 0.000 }
gfCNCPoint3[22276] = {X 129.0406, Y 10.4835, Z -4.6667, A 0.000, B 0.000, C 0.000 }
gfCNCPoint3[22277] = {X 129.1435, Y 9.5642, Z -4.6667, A 0.000, B 0.000, C 0.000 }
gfCNCPoint3[22278] = {X 129.4469, Y 8.6904, Z -4.6667, A 0.000, B 0.000, C 0.000 }
gfCNCPoint3[22279] = {X 129.9360, Y 7.9052, Z -4.6667, A 0.000, B 0.000, C 0.000 }
gfCNCPoint3[22280] = {X 130.5864, Y 7.2475, Z -4.6667, A 0.000, B 0.000, C 0.000 }
gfCNCPoint3[22281] = {X 131.3661, Y 6.7499, Z -4.6667, A 0.000, B 0.000, C 0.000 }
gfCNCPoint3[22282] = {X 132.2366, Y 6.4368, Z -4.6667, A 0.000, B 0.000, C 0.000 }
gfCNCPoint3[22283] = {X 133.1547, Y 6.3238, Z -4.6667, A 0.000, B 0.000, C 0.000 }
gfCNCPoint3[22284] = {X 133.8850, Y 6.3237, Z -4.6667, A 0.000, B 0.000, C 0.000 }
gfCNCPoint3[22285] = {X 134.6953, Y 6.4119, Z -4.6667, A 0.000, B 0.000, C 0.000 }
gfCNCPoint3[22286] = {X 135.4729, Y 6.6564, Z -4.6667, A 0.000, B 0.000, C 0.000 }
gfCNCPoint3[22287] = {X 136.1879, Y 7.0478, Z -4.6667, A 0.000, B 0.000, C 0.000 }
gfCNCPoint3[22288] = {X 136.8128, Y 7.5712, Z -4.6667, A 0.000, B 0.000, C 0.000 }
gfCNCPoint3[22289] = {X 137.3237, Y 8.2064, Z -4.6667, A 0.000, B 0.000, C 0.000 }
gfCNCPoint3[22290] = {X 155.1982, Y 8.2076, Z -4.6667, A 0.000, B 0.000, C 0.000 }
gfCNCPoint3[22291] = {X 155.7098, Y 7.5713, Z -4.6667, A 0.000, B 0.000, C 0.000 }
gfCNCPoint3[22292] = {X 156.3357, Y 7.0472, Z -4.6667, A 0.000, B 0.000, C 0.000 }
gfCNCPoint3[22293] = {X 157.0520, Y 6.6555, Z -4.6667, A 0.000, B 0.000, C 0.000 }
gfCNCPoint3[22294] = {X 157.8310, Y 6.4112, Z -4.6667, A 0.000, B 0.000, C 0.000 }
gfCNCPoint3[22295] = {X 158.6427, Y 6.3237, Z -4.6667, A 0.000, B 0.000, C 0.000 }
gfCNCPoint3[22296] = {X 159.3760, Y 6.3239, Z -4.6667, A 0.000, B 0.000, C 0.000 }
gfCNCPoint3[22297] = {X 160.2928, Y 6.4383, Z -4.6667, A 0.000, B 0.000, C 0.000 }
gfCNCPoint3[22298] = {X 161.1617, Y 6.7524, Z -4.6667, A 0.000, B 0.000, C 0.000 }
gfCNCPoint3[22299] = {X 161.9398, Y 7.2504, Z -4.6667, A 0.000, B 0.000, C 0.000 }
gfCNCPoint3[22300] = {X 162.5889, Y 7.9079, Z -4.6667, A 0.000, B 0.000, C 0.000 }
gfCNCPoint3[22301] = {X 163.0768, Y 8.6925, Z -4.6667, A 0.000, B 0.000, C 0.000 }
gfCNCPoint3[22302] = {X 163.3795, Y 9.5653, Z -4.6667, A 0.000, B 0.000, C 0.000 }
gfCNCPoint3[22303] = {X 163.4821, Y 10.4835, Z -4.6667, A 0.000, B 0.000, C 0.000 }
gfCNCPoint3[22304] = {X 163.4821, Y 17.4615, Z -4.6667, A 0.000, B 0.000, C 0.000 }
gfCNCPoint3[22305] = {X 163.3795, Y 18.3798, Z -4.6667, A 0.000, B 0.000, C 0.000 }
gfCNCPoint3[22306] = {X 163.0767, Y 19.2527, Z -4.6667, A 0.000, B 0.000, C 0.000 }
gfCNCPoint3[22307] = {X 162.5887, Y 20.0373, Z -4.6667, A 0.000, B 0.000, C 0.000 }
gfCNCPoint3[22308] = {X 161.9396, Y 20.6948, Z -4.6667, A 0.000, B 0.000, C 0.000 }
gfCNCPoint3[22309] = {X 161.1613, Y 21.1929, Z -4.6667, A 0.000, B 0.000, C 0.000 }
gfCNCPoint3[22310] = {X 160.2923, Y 21.5068, Z -4.6667, A 0.000, B 0.000, C 0.000 }
gfCNCPoint3[22311] = {X 159.3755, Y 21.6212, Z -4.6667, A 0.000, B 0.000, C 0.000 }
gfCNCPoint3[22312] = {X 158.6799, Y 21.6215, Z -4.6667, A 0.000, B 0.000, C 0.000 }
gfCNCPoint3[22313] = {X 157.8558, Y 21.5363, Z -4.6667, A 0.000, B 0.000, C 0.000 }
gfCNCPoint3[22314] = {X 157.0646, Y 21.2907, Z -4.6667, A 0.000, B 0.000, C 0.000 }
gfCNCPoint3[22315] = {X 156.3371, Y 20.8945, Z -4.6667, A 0.000, B 0.000, C 0.000 }
gfCNCPoint3[22316] = {X 155.7016, Y 20.3630, Z -4.6667, A 0.000, B 0.000, C 0.000 }
gfCNCPoint3[22317] = {X 155.1831, Y 19.7169, Z -4.6667, A 0.000, B 0.000, C 0.000 }
gfCNCPoint3[22318] = {X 152.1165, Y 19.7182, Z -4.6667, A 0.000, B 0.000, C 0.000 }
gfCNCPoint3[22319] = {X 152.1151, Y 40.9370, Z -4.6667, A 0.000, B 0.000, C 0.000 }
gfCNCPoint3[22320] = {X 152.6209, Y 41.4815, Z -4.6667, A 0.000, B 0.000, C 0.000 }
gfCNCPoint3[22321] = {X 152.7123, Y 41.5905, Z -4.6667, A 0.000, B 0.000, C 0.000 }
gfCNCPoint3[22322] = {X 153.2180, Y 42.3852, Z -4.6667, A 0.000, B 0.000, C 0.000 }
gfCNCPoint3[22323] = {X 153.5336, Y 43.2727, Z -4.6667, A 0.000, B 0.000, C 0.000 }
gfCNCPoint3[22324] = {X 153.6431, Y 44.2082, Z -4.6667, A 0.000, B 0.000, C 0.000 }
gfCNCPoint3[22325] = {X 153.6429, Y 45.0400, Z -4.6667, A 0.000, B 0.000, C 0.000 }
gfCNCPoint3[22326] = {X 153.5310, Y 45.9591, Z -4.6667, A 0.000, B 0.000, C 0.000 }
gfCNCPoint3[22327] = {X 153.2186, Y 46.8306, Z -4.6667, A 0.000, B 0.000, C 0.000 }
gfCNCPoint3[22328] = {X 152.7212, Y 47.6115, Z -4.6667, A 0.000, B 0.000, C 0.000 }
gfCNCPoint3[22329] = {X 152.0634, Y 48.2631, Z -4.6667, A 0.000, B 0.000, C 0.000 }
gfCNCPoint3[22330] = {X 151.2778, Y 48.7530, Z -4.6667, A 0.000, B 0.000, C 0.000 }
gfCNCPoint3[22331] = {X 150.4032, Y 49.0570, Z -4.6667, A 0.000, B 0.000, C 0.000 }
gfCNCPoint3[22332] = {X 149.4831, Y 49.1600, Z -4.6667, A 0.000, B 0.000, C 0.000 }
gfCNCPoint3[22333] = {X 143.0396, Y 49.1600, Z -4.6667, A 0.000, B 0.000, C 0.000 }
gfCNCPoint3[22334] = {X 142.1185, Y 49.0567, Z -4.6667, A 0.000, B 0.000, C 0.000 }
gfCNCPoint3[22335] = {X 141.2432, Y 48.7521, Z -4.6667, A 0.000, B 0.000, C 0.000 }
gfCNCPoint3[22336] = {X 140.4570, Y 48.2612, Z -4.6667, A 0.000, B 0.000, C 0.000 }
gfCNCPoint3[22337] = {X 139.7990, Y 47.6084, Z -4.6667, A 0.000, B 0.000, C 0.000 }
gfCNCPoint3[22338] = {X 139.3019, Y 46.8261, Z -4.6667, A 0.000, B 0.000, C 0.000 }
gfCNCPoint3[22339] = {X 138.9903, Y 45.9532, Z -4.6667, A 0.000, B 0.000, C 0.000 }
gfCNCPoint3[22340] = {X 138.8798, Y 45.0329, Z -4.6667, A 0.000, B 0.000, C 0.000 }
gfCNCPoint3[22341] = {X 138.8800, Y 44.1516, Z -4.6667, A 0.000, B 0.000, C 0.000 }
gfCNCPoint3[22342] = {X 138.9906, Y 43.2545, Z -4.6667, A 0.000, B 0.000, C 0.000 }
gfCNCPoint3[22343] = {X 139.2922, Y 42.4026, Z -4.6667, A 0.000, B 0.000, C 0.000 }
gfCNCPoint3[22344] = {X 139.7708, Y 41.6358, Z -4.6667, A 0.000, B 0.000, C 0.000 }
gfCNCPoint3[22345] = {X 140.4036, Y 40.9906, Z -4.6667, A 0.000, B 0.000, C 0.000 }
gfCNCPoint3[22346] = {X 140.4036, Y 30.3966, Z -4.6667, A 0.000, B 0.000, C 0.000 }
gfCNCPoint3[22347] = {X 136.4036, Y 30.3966, Z -4.6667, A 0.000, B 0.000, C 0.000 }
gfCNCPoint3[22348] = {X 140.4836, Y 30.3966, Z -4.6667, A 0.000, B 0.000, C 0.000 }
gfCNCPoint3[22349] = {X 140.4836, Y 19.6375, Z -4.6667, A 0.000, B 0.000, C 0.000 }
gfCNCPoint3[22350] = {X 137.2909, Y 19.6369, Z -4.6667, A 0.000, B 0.000, C 0.000 }
gfCNCPoint3[22351] = {X 137.2218, Y 19.7475, Z -4.6667, A 0.000, B 0.000, C 0.000 }
gfCNCPoint3[22352] = {X 136.5756, Y 20.4907, Z -4.6667, A 0.000, B 0.000, C 0.000 }
gfCNCPoint3[22353] = {X 135.7702, Y 21.0573, Z -4.6667, A 0.000, B 0.000, C 0.000 }
gfCNCPoint3[22354] = {X 134.8524, Y 21.4145, Z -4.6667, A 0.000, B 0.000, C 0.000 }
gfCNCPoint3[22355] = {X 133.8758, Y 21.5414, Z -4.6667, A 0.000, B 0.000, C 0.000 }
gfCNCPoint3[22356] = {X 133.2006, Y 21.5415, Z -4.6667, A 0.000, B 0.000, C 0.000 }
gfCNCPoint3[22357] = {X 132.2928, Y 21.4392, Z -4.6667, A 0.000, B 0.000, C 0.000 }
gfCNCPoint3[22358] = {X 131.4304, Y 21.1375, Z -4.6667, A 0.000, B 0.000, C 0.000 }
gfCNCPoint3[22359] = {X 130.6568, Y 20.6514, Z -4.6667, A 0.000, B 0.000, C 0.000 }
gfCNCPoint3[22360] = {X 130.0108, Y 20.0054, Z -4.6667, A 0.000, B 0.000, C 0.000 }
gfCNCPoint3[22361] = {X 129.5247, Y 19.2318, Z -4.6667, A 0.000, B 0.000, C 0.000 }
gfCNCPoint3[22362] = {X 129.2229, Y 18.3694, Z -4.6667, A 0.000, B 0.000, C 0.000 }
gfCNCPoint3[22363] = {X 129.1206, Y 17.4615, Z -4.6667, A 0.000, B 0.000, C 0.000 }
gfCNCPoint3[22364] = {X 129.1206, Y 10.4835, Z -4.6667, A 0.000, B 0.000, C 0.000 }
gfCNCPoint3[22365] = {X 129.2215, Y 9.5820, Z -4.6667, A 0.000, B 0.000, C 0.000 }
gfCNCPoint3[22366] = {X 129.5191, Y 8.7250, Z -4.6667, A 0.000, B 0.000, C 0.000 }
gfCNCPoint3[22367] = {X 129.9986, Y 7.9550, Z -4.6667, A 0.000, B 0.000, C 0.000 }
gfCNCPoint3[22368] = {X 130.6365, Y 7.3099, Z -4.6667, A 0.000, B 0.000, C 0.000 }
gfCNCPoint3[22369] = {X 131.4011, Y 6.8218, Z -4.6667, A 0.000, B 0.000, C 0.000 }
gfCNCPoint3[22370] = {X 132.2547, Y 6.5147, Z -4.6667, A 0.000, B 0.000, C 0.000 }
gfCNCPoint3[22371] = {X 133.1551, Y 6.4038, Z -4.6667, A 0.000, B 0.000, C 0.000 }
gfCNCPoint3[22372] = {X 133.8841, Y 6.4037, Z -4.6667, A 0.000, B 0.000, C 0.000 }
gfCNCPoint3[22373] = {X 134.6873, Y 6.4920, Z -4.6667, A 0.000, B 0.000, C 0.000 }
gfCNCPoint3[22374] = {X 135.4574, Y 6.7368, Z -4.6667, A 0.000, B 0.000, C 0.000 }
gfCNCPoint3[22375] = {X 136.1641, Y 7.1286, Z -4.6667, A 0.000, B 0.000, C 0.000 }
gfCNCPoint3[22376] = {X 136.7797, Y 7.6519, Z -4.6667, A 0.000, B 0.000, C 0.000 }
gfCNCPoint3[22377] = {X 137.2802, Y 8.2864, Z -4.6667, A 0.000, B 0.000, C 0.000 }
gfCNCPoint3[22378] = {X 155.2418, Y 8.2876, Z -4.6667, A 0.000, B 0.000, C 0.000 }
gfCNCPoint3[22379] = {X 155.2872, Y 8.2180, Z -4.6667, A 0.000, B 0.000, C 0.000 }
gfCNCPoint3[22380] = {X 155.3340, Y 8.1494, Z -4.6667, A 0.000, B 0.000, C 0.000 }
gfCNCPoint3[22381] = {X 155.9792, Y 7.4258, Z -4.6667, A 0.000, B 0.000, C 0.000 }
gfCNCPoint3[22382] = {X 156.7768, Y 6.8748, Z -4.6667, A 0.000, B 0.000, C 0.000 }
gfCNCPoint3[22383] = {X 157.6819, Y 6.5276, Z -4.6667, A 0.000, B 0.000, C 0.000 }
gfCNCPoint3[22384] = {X 158.6434, Y 6.4037, Z -4.6667, A 0.000, B 0.000, C 0.000 }
gfCNCPoint3[22385] = {X 159.3750, Y 6.4039, Z -4.6667, A 0.000, B 0.000, C 0.000 }
gfCNCPoint3[22386] = {X 160.2741, Y 6.5161, Z -4.6667, A 0.000, B 0.000, C 0.000 }
gfCNCPoint3[22387] = {X 161.1263, Y 6.8241, Z -4.6667, A 0.000, B 0.000, C 0.000 }
gfCNCPoint3[22388] = {X 161.8895, Y 7.3126, Z -4.6667, A 0.000, B 0.000, C 0.000 }
gfCNCPoint3[22389] = {X 162.5260, Y 7.9574, Z -4.6667, A 0.000, B 0.000, C 0.000 }
gfCNCPoint3[22390] = {X 163.0046, Y 8.7269, Z -4.6667, A 0.000, B 0.000, C 0.000 }
gfCNCPoint3[22391] = {X 163.3015, Y 9.5830, Z -4.6667, A 0.000, B 0.000, C 0.000 }
gfCNCPoint3[22392] = {X 163.4021, Y 10.4835, Z -4.6667, A 0.000, B 0.000, C 0.000 }
gfCNCPoint3[22393] = {X 163.4021, Y 17.4615, Z -4.6667, A 0.000, B 0.000, C 0.000 }
gfCNCPoint3[22394] = {X 163.3015, Y 18.3621, Z -4.6667, A 0.000, B 0.000, C 0.000 }
gfCNCPoint3[22395] = {X 163.0046, Y 19.2182, Z -4.6667, A 0.000, B 0.000, C 0.000 }
gfCNCPoint3[22396] = {X 162.5260, Y 19.9876, Z -4.6667, A 0.000, B 0.000, C 0.000 }
gfCNCPoint3[22397] = {X 161.8895, Y 20.6325, Z -4.6667, A 0.000, B 0.000, C 0.000 }
gfCNCPoint3[22398] = {X 161.1263, Y 21.1209, Z -4.6667, A 0.000, B 0.000, C 0.000 }
gfCNCPoint3[22399] = {X 160.2741, Y 21.4289, Z -4.6667, A 0.000, B 0.000, C 0.000 }
gfCNCPoint3[22400] = {X 159.3750, Y 21.5412, Z -4.6667, A 0.000, B 0.000, C 0.000 }
gfCNCPoint3[22401] = {X 158.6802, Y 21.5415, Z -4.6667, A 0.000, B 0.000, C 0.000 }
gfCNCPoint3[22402] = {X 157.8634, Y 21.4562, Z -4.6667, A 0.000, B 0.000, C 0.000 }
gfCNCPoint3[22403] = {X 157.0798, Y 21.2103, Z -4.6667, A 0.000, B 0.000, C 0.000 }
gfCNCPoint3[22404] = {X 156.3607, Y 20.8137, Z -4.6667, A 0.000, B 0.000, C 0.000 }
gfCNCPoint3[22405] = {X 155.7347, Y 20.2822, Z -4.6667, A 0.000, B 0.000, C 0.000 }
gfCNCPoint3[22406] = {X 155.2267, Y 19.6369, Z -4.6667, A 0.000, B 0.000, C 0.000 }
gfCNCPoint3[22407] = {X 152.0365, Y 19.6382, Z -4.6667, A 0.000, B 0.000, C 0.000 }
gfCNCPoint3[22408] = {X 152.0351, Y 40.9684, Z -4.6667, A 0.000, B 0.000, C 0.000 }
gfCNCPoint3[22409] = {X 152.5609, Y 41.5345, Z -4.6667, A 0.000, B 0.000, C 0.000 }
gfCNCPoint3[22410] = {X 152.6505, Y 41.6414, Z -4.6667, A 0.000, B 0.000, C 0.000 }
gfCNCPoint3[22411] = {X 153.1463, Y 42.4207, Z -4.6667, A 0.000, B 0.000, C 0.000 }
gfCNCPoint3[22412] = {X 153.4557, Y 43.2911, Z -4.6667, A 0.000, B 0.000, C 0.000 }
gfCNCPoint3[22413] = {X 153.5631, Y 44.2086, Z -4.6667, A 0.000, B 0.000, C 0.000 }
gfCNCPoint3[22414] = {X 153.5629, Y 45.0392, Z -4.6667, A 0.000, B 0.000, C 0.000 }
gfCNCPoint3[22415] = {X 153.4532, Y 45.9406, Z -4.6667, A 0.000, B 0.000, C 0.000 }
gfCNCPoint3[22416] = {X 153.1468, Y 46.7954, Z -4.6667, A 0.000, B 0.000, C 0.000 }
gfCNCPoint3[22417] = {X 152.6589, Y 47.5613, Z -4.6667, A 0.000, B 0.000, C 0.000 }
gfCNCPoint3[22418] = {X 152.0138, Y 48.2003, Z -4.6667, A 0.000, B 0.000, C 0.000 }
gfCNCPoint3[22419] = {X 151.2432, Y 48.6808, Z -4.6667, A 0.000, B 0.000, C 0.000 }
gfCNCPoint3[22420] = {X 150.3855, Y 48.9789, Z -4.6667, A 0.000, B 0.000, C 0.000 }
gfCNCPoint3[22421] = {X 149.4831, Y 49.0800, Z -4.6667, A 0.000, B 0.000, C 0.000 }
gfCNCPoint3[22422] = {X 143.0396, Y 49.0800, Z -4.6667, A 0.000, B 0.000, C 0.000 }
gfCNCPoint3[22423] = {X 142.1362, Y 48.9787, Z -4.6667, A 0.000, B 0.000, C 0.000 }
gfCNCPoint3[22424] = {X 141.2777, Y 48.6799, Z -4.6667, A 0.000, B 0.000, C 0.000 }
gfCNCPoint3[22425] = {X 140.5066, Y 48.1985, Z -4.6667, A 0.000, B 0.000, C 0.000 }
gfCNCPoint3[22426] = {X 139.8613, Y 47.5582, Z -4.6667, A 0.000, B 0.000, C 0.000 }
gfCNCPoint3[22427] = {X 139.3737, Y 46.7910, Z -4.6667, A 0.000, B 0.000, C 0.000 }
gfCNCPoint3[22428] = {X 139.0682, Y 45.9349, Z -4.6667, A 0.000, B 0.000, C 0.000 }
gfCNCPoint3[22429] = {X 138.9598, Y 45.0323, Z -4.6667, A 0.000, B 0.000, C 0.000 }
gfCNCPoint3[22430] = {X 138.9600, Y 44.1527, Z -4.6667, A 0.000, B 0.000, C 0.000 }
gfCNCPoint3[22431] = {X 139.0706, Y 43.2637, Z -4.6667, A 0.000, B 0.000, C 0.000 }
gfCNCPoint3[22432] = {X 139.3725, Y 42.4203, Z -4.6667, A 0.000, B 0.000, C 0.000 }
gfCNCPoint3[22433] = {X 139.8512, Y 41.6631, Z -4.6667, A 0.000, B 0.000, C 0.000 }
gfCNCPoint3[22434] = {X 140.4836, Y 41.0287, Z -4.6667, A 0.000, B 0.000, C 0.000 }
gfCNCPoint3[22435] = {X 140.4836, Y 30.3966, Z -4.6667, A 0.000, B 0.000, C 0.000 }
gfCNCPoint3[22436] = {X 136.4836, Y 30.3966, Z -4.6667, A 0.000, B 0.000, C 0.000 }
gfCNCPoint3[22437] = {X 140.5636, Y 30.3966, Z -4.6667, A 0.000, B 0.000, C 0.000 }
gfCNCPoint3[22438] = {X 140.5636, Y 19.9575, Z -4.6667, A 0.000, B 0.000, C 0.000 }
gfCNCPoint3[22439] = {X 140.5643, Y 19.5575, Z -4.6667, A 0.000, B 0.000, C 0.000 }
gfCNCPoint3[22440] = {X 137.2663, Y 19.5569, Z -4.6667, A 0.000, B 0.000, C 0.000 }
gfCNCPoint3[22441] = {X 137.2441, Y 19.5609, Z -4.6667, A 0.000, B 0.000, C 0.000 }
gfCNCPoint3[22442] = {X 137.1368, Y 19.7301, Z -4.6667, A 0.000, B 0.000, C 0.000 }
gfCNCPoint3[22443] = {X 136.4973, Y 20.4533, Z -4.6667, A 0.000, B 0.000, C 0.000 }
gfCNCPoint3[22444] = {X 135.7032, Y 21.0023, Z -4.6667, A 0.000, B 0.000, C 0.000 }
gfCNCPoint3[22445] = {X 134.8006, Y 21.3451, Z -4.6667, A 0.000, B 0.000, C 0.000 }
gfCNCPoint3[22446] = {X 133.8422, Y 21.4615, Z -4.6667, A 0.000, B 0.000, C 0.000 }
gfCNCPoint3[22447] = {X 133.2006, Y 21.4615, Z -4.6667, A 0.000, B 0.000, C 0.000 }
gfCNCPoint3[22448] = {X 132.3106, Y 21.3613, Z -4.6667, A 0.000, B 0.000, C 0.000 }
gfCNCPoint3[22449] = {X 131.4651, Y 21.0654, Z -4.6667, A 0.000, B 0.000, C 0.000 }
gfCNCPoint3[22450] = {X 130.7067, Y 20.5889, Z -4.6667, A 0.000, B 0.000, C 0.000 }
gfCNCPoint3[22451] = {X 130.0733, Y 19.9555, Z -4.6667, A 0.000, B 0.000, C 0.000 }
gfCNCPoint3[22452] = {X 129.5968, Y 19.1971, Z -4.6667, A 0.000, B 0.000, C 0.000 }
gfCNCPoint3[22453] = {X 129.3009, Y 18.3516, Z -4.6667, A 0.000, B 0.000, C 0.000 }
gfCNCPoint3[22454] = {X 129.2006, Y 17.4615, Z -4.6667, A 0.000, B 0.000, C 0.000 }
gfCNCPoint3[22455] = {X 129.2006, Y 10.4835, Z -4.6667, A 0.000, B 0.000, C 0.000 }
gfCNCPoint3[22456] = {X 129.3009, Y 9.5934, Z -4.6667, A 0.000, B 0.000, C 0.000 }
gfCNCPoint3[22457] = {X 129.5968, Y 8.7480, Z -4.6667, A 0.000, B 0.000, C 0.000 }
gfCNCPoint3[22458] = {X 130.0733, Y 7.9896, Z -4.6667, A 0.000, B 0.000, C 0.000 }
gfCNCPoint3[22459] = {X 130.7067, Y 7.3562, Z -4.6667, A 0.000, B 0.000, C 0.000 }
gfCNCPoint3[22460] = {X 131.4651, Y 6.8796, Z -4.6667, A 0.000, B 0.000, C 0.000 }
gfCNCPoint3[22461] = {X 132.3106, Y 6.5838, Z -4.6667, A 0.000, B 0.000, C 0.000 }
gfCNCPoint3[22462] = {X 133.2007, Y 6.4835, Z -4.6667, A 0.000, B 0.000, C 0.000 }
gfCNCPoint3[22463] = {X 133.8833, Y 6.4837, Z -4.6667, A 0.000, B 0.000, C 0.000 }
gfCNCPoint3[22464] = {X 134.6793, Y 6.5721, Z -4.6667, A 0.000, B 0.000, C 0.000 }
gfCNCPoint3[22465] = {X 135.4418, Y 6.8172, Z -4.6667, A 0.000, B 0.000, C 0.000 }
gfCNCPoint3[22466] = {X 136.1401, Y 7.2093, Z -4.6667, A 0.000, B 0.000, C 0.000 }
gfCNCPoint3[22467] = {X 136.7463, Y 7.7327, Z -4.6667, A 0.000, B 0.000, C 0.000 }
gfCNCPoint3[22468] = {X 137.2361, Y 8.3664, Z -4.6667, A 0.000, B 0.000, C 0.000 }
gfCNCPoint3[22469] = {X 155.2276, Y 8.3664, Z -4.6667, A 0.000, B 0.000, C 0.000 }
gfCNCPoint3[22470] = {X 155.2814, Y 8.3748, Z -4.6667, A 0.000, B 0.000, C 0.000 }
gfCNCPoint3[22471] = {X 155.3393, Y 8.2842, Z -4.6667, A 0.000, B 0.000, C 0.000 }
gfCNCPoint3[22472] = {X 155.3996, Y 8.1952, Z -4.6667, A 0.000, B 0.000, C 0.000 }
gfCNCPoint3[22473] = {X 156.0390, Y 7.4797, Z -4.6667, A 0.000, B 0.000, C 0.000 }
gfCNCPoint3[22474] = {X 156.8303, Y 6.9371, Z -4.6667, A 0.000, B 0.000, C 0.000 }
gfCNCPoint3[22475] = {X 157.7280, Y 6.5986, Z -4.6667, A 0.000, B 0.000, C 0.000 }
gfCNCPoint3[22476] = {X 158.6806, Y 6.4835, Z -4.6667, A 0.000, B 0.000, C 0.000 }
gfCNCPoint3[22477] = {X 159.3739, Y 6.4839, Z -4.6667, A 0.000, B 0.000, C 0.000 }
gfCNCPoint3[22478] = {X 160.2554, Y 6.5939, Z -4.6667, A 0.000, B 0.000, C 0.000 }
gfCNCPoint3[22479] = {X 161.0909, Y 6.8959, Z -4.6667, A 0.000, B 0.000, C 0.000 }
gfCNCPoint3[22480] = {X 161.8391, Y 7.3747, Z -4.6667, A 0.000, B 0.000, C 0.000 }
gfCNCPoint3[22481] = {X 162.4632, Y 8.0070, Z -4.6667, A 0.000, B 0.000, C 0.000 }
gfCNCPoint3[22482] = {X 162.9324, Y 8.7613, Z -4.6667, A 0.000, B 0.000, C 0.000 }
gfCNCPoint3[22483] = {X 163.2234, Y 9.6007, Z -4.6667, A 0.000, B 0.000, C 0.000 }
gfCNCPoint3[22484] = {X 163.3221, Y 10.4835, Z -4.6667, A 0.000, B 0.000, C 0.000 }
gfCNCPoint3[22485] = {X 163.3221, Y 17.4615, Z -4.6667, A 0.000, B 0.000, C 0.000 }
gfCNCPoint3[22486] = {X 163.2218, Y 18.3516, Z -4.6667, A 0.000, B 0.000, C 0.000 }
gfCNCPoint3[22487] = {X 162.9260, Y 19.1971, Z -4.6667, A 0.000, B 0.000, C 0.000 }
gfCNCPoint3[22488] = {X 162.4494, Y 19.9555, Z -4.6667, A 0.000, B 0.000, C 0.000 }
gfCNCPoint3[22489] = {X 161.8160, Y 20.5889, Z -4.6667, A 0.000, B 0.000, C 0.000 }
gfCNCPoint3[22490] = {X 161.0576, Y 21.0654, Z -4.6667, A 0.000, B 0.000, C 0.000 }
gfCNCPoint3[22491] = {X 160.2121, Y 21.3613, Z -4.6667, A 0.000, B 0.000, C 0.000 }
gfCNCPoint3[22492] = {X 159.3221, Y 21.4615, Z -4.6667, A 0.000, B 0.000, C 0.000 }
gfCNCPoint3[22493] = {X 158.6805, Y 21.4615, Z -4.6667, A 0.000, B 0.000, C 0.000 }
gfCNCPoint3[22494] = {X 157.8710, Y 21.3760, Z -4.6667, A 0.000, B 0.000, C 0.000 }
gfCNCPoint3[22495] = {X 157.0952, Y 21.1298, Z -4.6667, A 0.000, B 0.000, C 0.000 }
gfCNCPoint3[22496] = {X 156.3846, Y 20.7328, Z -4.6667, A 0.000, B 0.000, C 0.000 }
gfCNCPoint3[22497] = {X 155.7681, Y 20.2013, Z -4.6667, A 0.000, B 0.000, C 0.000 }
gfCNCPoint3[22498] = {X 155.2709, Y 19.5569, Z -4.6667, A 0.000, B 0.000, C 0.000 }
gfCNCPoint3[22499] = {X 151.9565, Y 19.5583, Z -4.6667, A 0.000, B 0.000, C 0.000 }
gfCNCPoint3[22500] = {X 151.9551, Y 40.9999, Z -4.6667, A 0.000, B 0.000, C 0.000 }
gfCNCPoint3[22501] = {X 152.5009, Y 41.5875, Z -4.6667, A 0.000, B 0.000, C 0.000 }
gfCNCPoint3[22502] = {X 152.5888, Y 41.6922, Z -4.6667, A 0.000, B 0.000, C 0.000 }
gfCNCPoint3[22503] = {X 153.0747, Y 42.4563, Z -4.6667, A 0.000, B 0.000, C 0.000 }
gfCNCPoint3[22504] = {X 153.3779, Y 43.3095, Z -4.6667, A 0.000, B 0.000, C 0.000 }
gfCNCPoint3[22505] = {X 153.4831, Y 44.2089, Z -4.6667, A 0.000, B 0.000, C 0.000 }
gfCNCPoint3[22506] = {X 153.4829, Y 45.0384, Z -4.6667, A 0.000, B 0.000, C 0.000 }
gfCNCPoint3[22507] = {X 153.3753, Y 45.9222, Z -4.6667, A 0.000, B 0.000, C 0.000 }
gfCNCPoint3[22508] = {X 153.0750, Y 46.7602, Z -4.6667, A 0.000, B 0.000, C 0.000 }
gfCNCPoint3[22509] = {X 152.5967, Y 47.5111, Z -4.6667, A 0.000, B 0.000, C 0.000 }
gfCNCPoint3[22510] = {X 151.9642, Y 48.1376, Z -4.6667, A 0.000, B 0.000, C 0.000 }
gfCNCPoint3[22511] = {X 151.2087, Y 48.6086, Z -4.6667, A 0.000, B 0.000, C 0.000 }
gfCNCPoint3[22512] = {X 150.3678, Y 48.9009, Z -4.6667, A 0.000, B 0.000, C 0.000 }
gfCNCPoint3[22513] = {X 149.4831, Y 49.0000, Z -4.6667, A 0.000, B 0.000, C 0.000 }
gfCNCPoint3[22514] = {X 143.0396, Y 49.0000, Z -4.6667, A 0.000, B 0.000, C 0.000 }
gfCNCPoint3[22515] = {X 142.1495, Y 48.8997, Z -4.6667, A 0.000, B 0.000, C 0.000 }
gfCNCPoint3[22516] = {X 141.3041, Y 48.6039, Z -4.6667, A 0.000, B 0.000, C 0.000 }
gfCNCPoint3[22517] = {X 140.5457, Y 48.1273, Z -4.6667, A 0.000, B 0.000, C 0.000 }
gfCNCPoint3[22518] = {X 139.9123, Y 47.4939, Z -4.6667, A 0.000, B 0.000, C 0.000 }
gfCNCPoint3[22519] = {X 139.4357, Y 46.7355, Z -4.6667, A 0.000, B 0.000, C 0.000 }
gfCNCPoint3[22520] = {X 139.1399, Y 45.8901, Z -4.6667, A 0.000, B 0.000, C 0.000 }
gfCNCPoint3[22521] = {X 139.0396, Y 45.0000, Z -4.6667, A 0.000, B 0.000, C 0.000 }
gfCNCPoint3[22522] = {X 139.0400, Y 44.1538, Z -4.6667, A 0.000, B 0.000, C 0.000 }
gfCNCPoint3[22523] = {X 139.1506, Y 43.2730, Z -4.6667, A 0.000, B 0.000, C 0.000 }
gfCNCPoint3[22524] = {X 139.4528, Y 42.4382, Z -4.6667, A 0.000, B 0.000, C 0.000 }
gfCNCPoint3[22525] = {X 139.9317, Y 41.6907, Z -4.6667, A 0.000, B 0.000, C 0.000 }
gfCNCPoint3[22526] = {X 140.5636, Y 41.0672, Z -4.6667, A 0.000, B 0.000, C 0.000 }
gfCNCPoint3[22527] = {X 140.5636, Y 30.3966, Z -4.6667, A 0.000, B 0.000, C 0.000 }
gfCNCPoint3[22528] = {X 136.4836, Y 30.3966, Z -4.6667, A 0.000, B 0.000, C 0.000 }
gfCNCPoint3[22529] = {X 136.4836, Y 30.3966, Z -1.6667, A 0.000, B 0.000, C 0.000 }
gfCNCPoint3[22530] = {X 136.4836, Y 30.3966, Z 11.0000, A 0.000, B 0.000, C 0.000 }
gfCNCPoint3[22531] = {X 137.6635, Y 74.8927, Z 11.0000, A 0.000, B 0.000, C 0.000 }
gfCNCPoint3[22532] = {X 137.6635, Y 74.8927, Z -1.6667, A 0.000, B 0.000, C 0.000 }
gfCNCPoint3[22533] = {X 137.6635, Y 74.8927, Z -4.6667, A 0.000, B 0.000, C 0.000 }
gfCNCPoint3[22534] = {X 140.6802, Y 77.6397, Z -4.6667, A 0.000, B 0.000, C 0.000 }
gfCNCPoint3[22535] = {X 155.6324, Y 61.2201, Z -4.6667, A 0.000, B 0.000, C 0.000 }
gfCNCPoint3[22536] = {X 155.2774, Y 60.5144, Z -4.6667, A 0.000, B 0.000, C 0.000 }
gfCNCPoint3[22537] = {X 155.0568, Y 59.7558, Z -4.6667, A 0.000, B 0.000, C 0.000 }
gfCNCPoint3[22538] = {X 154.9781, Y 58.9697, Z -4.6667, A 0.000, B 0.000, C 0.000 }
gfCNCPoint3[22539] = {X 154.9780, Y 58.0000, Z -4.6667, A 0.000, B 0.000, C 0.000 }
gfCNCPoint3[22540] = {X 155.0863, Y 57.0387, Z -4.6667, A 0.000, B 0.000, C 0.000 }
gfCNCPoint3[22541] = {X 155.4058, Y 56.1256, Z -4.6667, A 0.000, B 0.000, C 0.000 }
gfCNCPoint3[22542] = {X 155.9204, Y 55.3065, Z -4.6667, A 0.000, B 0.000, C 0.000 }
gfCNCPoint3[22543] = {X 156.6045, Y 54.6225, Z -4.6667, A 0.000, B 0.000, C 0.000 }
gfCNCPoint3[22544] = {X 157.4236, Y 54.1078, Z -4.6667, A 0.000, B 0.000, C 0.000 }
gfCNCPoint3[22545] = {X 158.3367, Y 53.7883, Z -4.6667, A 0.000, B 0.000, C 0.000 }
gfCNCPoint3[22546] = {X 159.2980, Y 53.6800, Z -4.6667, A 0.000, B 0.000, C 0.000 }
gfCNCPoint3[22547] = {X 178.5335, Y 53.6800, Z -4.6667, A 0.000, B 0.000, C 0.000 }
gfCNCPoint3[22548] = {X 179.4948, Y 53.7883, Z -4.6667, A 0.000, B 0.000, C 0.000 }
gfCNCPoint3[22549] = {X 180.4079, Y 54.1078, Z -4.6667, A 0.000, B 0.000, C 0.000 }
gfCNCPoint3[22550] = {X 181.2270, Y 54.6225, Z -4.6667, A 0.000, B 0.000, C 0.000 }
gfCNCPoint3[22551] = {X 181.9110, Y 55.3065, Z -4.6667, A 0.000, B 0.000, C 0.000 }
gfCNCPoint3[22552] = {X 182.4257, Y 56.1256, Z -4.6667, A 0.000, B 0.000, C 0.000 }
gfCNCPoint3[22553] = {X 182.7452, Y 57.0387, Z -4.6667, A 0.000, B 0.000, C 0.000 }
gfCNCPoint3[22554] = {X 182.8535, Y 58.0000, Z -4.6667, A 0.000, B 0.000, C 0.000 }
gfCNCPoint3[22555] = {X 182.8535, Y 58.9342, Z -4.6667, A 0.000, B 0.000, C 0.000 }
gfCNCPoint3[22556] = {X 182.7808, Y 59.7233, Z -4.6667, A 0.000, B 0.000, C 0.000 }
gfCNCPoint3[22557] = {X 182.5652, Y 60.4858, Z -4.6667, A 0.000, B 0.000, C 0.000 }
gfCNCPoint3[22558] = {X 182.2139, Y 61.1961, Z -4.6667, A 0.000, B 0.000, C 0.000 }
gfCNCPoint3[22559] = {X 209.4788, Y 90.9541, Z -4.6667, A 0.000, B 0.000, C 0.000 }
gfCNCPoint3[22560] = {X 210.1359, Y 91.6209, Z -4.6667, A 0.000, B 0.000, C 0.000 }
gfCNCPoint3[22561] = {X 210.8398, Y 92.2380, Z -4.6667, A 0.000, B 0.000, C 0.000 }
gfCNCPoint3[22562] = {X 211.1139, Y 92.4114, Z -4.6667, A 0.000, B 0.000, C 0.000 }
gfCNCPoint3[22563] = {X 211.4211, Y 92.5152, Z -4.6667, A 0.000, B 0.000, C 0.000 }
gfCNCPoint3[22564] = {X 213.4040, Y 92.8245, Z -4.6667, A 0.000, B 0.000, C 0.000 }
gfCNCPoint3[22565] = {X 214.4546, Y 92.7358, Z -4.6667, A 0.000, B 0.000, C 0.000 }
gfCNCPoint3[22566] = {X 215.5072, Y 92.6756, Z -4.6667, A 0.000, B 0.000, C 0.000 }
gfCNCPoint3[22567] = {X 216.1773, Y 92.6024, Z -4.6667, A 0.000, B 0.000, C 0.000 }
gfCNCPoint3[22568] = {X 216.8225, Y 92.4074, Z -4.6667, A 0.000, B 0.000, C 0.000 }
gfCNCPoint3[22569] = {X 217.4210, Y 92.0971, Z -4.6667, A 0.000, B 0.000, C 0.000 }
gfCNCPoint3[22570] = {X 222.9613, Y 88.5216, Z -4.6667, A 0.000, B 0.000, C 0.000 }
gfCNCPoint3[22571] = {X 245.8281, Y 73.8996, Z -4.6667, A 0.000, B 0.000, C 0.000 }
gfCNCPoint3[22572] = {X 221.6305, Y 64.4037, Z -4.6667, A 0.000, B 0.000, C 0.000 }
gfCNCPoint3[22573] = {X 219.8631, Y 63.8121, Z -4.6667, A 0.000, B 0.000, C 0.000 }
gfCNCPoint3[22574] = {X 218.0397, Y 63.4263, Z -4.6667, A 0.000, B 0.000, C 0.000 }
gfCNCPoint3[22575] = {X 216.1841, Y 63.2516, Z -4.6667, A 0.000, B 0.000, C 0.000 }
gfCNCPoint3[22576] = {X 215.2523, Y 63.1173, Z -4.6667, A 0.000, B 0.000, C 0.000 }
gfCNCPoint3[22577] = {X 214.3717, Y 62.7843, Z -4.6667, A 0.000, B 0.000, C 0.000 }
gfCNCPoint3[22578] = {X 213.5841, Y 62.2684, Z -4.6667, A 0.000, B 0.000, C 0.000 }
gfCNCPoint3[22579] = {X 212.9270, Y 61.5942, Z -4.6667, A 0.000, B 0.000, C 0.000 }
gfCNCPoint3[22580] = {X 212.4315, Y 60.7936, Z -4.6667, A 0.000, B 0.000, C 0.000 }
gfCNCPoint3[22581] = {X 212.1213, Y 59.9047, Z -4.6667, A 0.000, B 0.000, C 0.000 }
gfCNCPoint3[22582] = {X 212.0110, Y 58.9697, Z -4.6667, A 0.000, B 0.000, C 0.000 }
gfCNCPoint3[22583] = {X 212.0108, Y 58.0000, Z -4.6667, A 0.000, B 0.000, C 0.000 }
gfCNCPoint3[22584] = {X 212.1191, Y 57.0387, Z -4.6667, A 0.000, B 0.000, C 0.000 }
gfCNCPoint3[22585] = {X 212.4386, Y 56.1256, Z -4.6667, A 0.000, B 0.000, C 0.000 }
gfCNCPoint3[22586] = {X 212.9533, Y 55.3065, Z -4.6667, A 0.000, B 0.000, C 0.000 }
gfCNCPoint3[22587] = {X 213.6373, Y 54.6225, Z -4.6667, A 0.000, B 0.000, C 0.000 }
gfCNCPoint3[22588] = {X 214.4564, Y 54.1078, Z -4.6667, A 0.000, B 0.000, C 0.000 }
gfCNCPoint3[22589] = {X 215.3695, Y 53.7883, Z -4.6667, A 0.000, B 0.000, C 0.000 }
gfCNCPoint3[22590] = {X 216.3308, Y 53.6800, Z -4.6667, A 0.000, B 0.000, C 0.000 }
gfCNCPoint3[22591] = {X 237.2617, Y 53.6800, Z -4.6667, A 0.000, B 0.000, C 0.000 }
gfCNCPoint3[22592] = {X 238.2230, Y 53.7883, Z -4.6667, A 0.000, B 0.000, C 0.000 }
gfCNCPoint3[22593] = {X 239.1361, Y 54.1078, Z -4.6667, A 0.000, B 0.000, C 0.000 }
gfCNCPoint3[22594] = {X 239.9552, Y 54.6225, Z -4.6667, A 0.000, B 0.000, C 0.000 }
gfCNCPoint3[22595] = {X 240.6392, Y 55.3065, Z -4.6667, A 0.000, B 0.000, C 0.000 }
gfCNCPoint3[22596] = {X 241.1539, Y 56.1256, Z -4.6667, A 0.000, B 0.000, C 0.000 }
gfCNCPoint3[22597] = {X 241.4734, Y 57.0387, Z -4.6667, A 0.000, B 0.000, C 0.000 }
gfCNCPoint3[22598] = {X 241.5817, Y 58.0000, Z -4.6667, A 0.000, B 0.000, C 0.000 }
gfCNCPoint3[22599] = {X 241.5817, Y 58.2323, Z -4.6667, A 0.000, B 0.000, C 0.000 }
gfCNCPoint3[22600] = {X 248.1138, Y 60.7793, Z -4.6667, A 0.000, B 0.000, C 0.000 }
gfCNCPoint3[22601] = {X 275.6329, Y 71.7021, Z -4.6667, A 0.000, B 0.000, C 0.000 }
gfCNCPoint3[22602] = {X 275.6340, Y 63.2124, Z -4.6667, A 0.000, B 0.000, C 0.000 }
gfCNCPoint3[22603] = {X 274.7823, Y 63.0033, Z -4.6667, A 0.000, B 0.000, C 0.000 }
gfCNCPoint3[22604] = {X 273.9903, Y 62.6265, Z -4.6667, A 0.000, B 0.000, C 0.000 }
gfCNCPoint3[22605] = {X 273.2908, Y 62.0976, Z -4.6667, A 0.000, B 0.000, C 0.000 }
gfCNCPoint3[22606] = {X 272.7125, Y 61.4383, Z -4.6667, A 0.000, B 0.000, C 0.000 }
gfCNCPoint3[22607] = {X 272.2793, Y 60.6757, Z -4.6667, A 0.000, B 0.000, C 0.000 }
gfCNCPoint3[22608] = {X 272.0091, Y 59.8414, Z -4.6667, A 0.000, B 0.000, C 0.000 }
gfCNCPoint3[22609] = {X 271.9128, Y 58.9697, Z -4.6667, A 0.000, B 0.000, C 0.000 }
gfCNCPoint3[22610] = {X 271.9127, Y 58.0000, Z -4.6667, A 0.000, B 0.000, C 0.000 }
gfCNCPoint3[22611] = {X 272.0210, Y 57.0387, Z -4.6667, A 0.000, B 0.000, C 0.000 }
gfCNCPoint3[22612] = {X 272.3405, Y 56.1256, Z -4.6667, A 0.000, B 0.000, C 0.000 }
gfCNCPoint3[22613] = {X 272.8552, Y 55.3065, Z -4.6667, A 0.000, B 0.000, C 0.000 }
gfCNCPoint3[22614] = {X 273.5392, Y 54.6225, Z -4.6667, A 0.000, B 0.000, C 0.000 }
gfCNCPoint3[22615] = {X 274.3583, Y 54.1078, Z -4.6667, A 0.000, B 0.000, C 0.000 }
gfCNCPoint3[22616] = {X 275.2714, Y 53.7883, Z -4.6667, A 0.000, B 0.000, C 0.000 }
gfCNCPoint3[22617] = {X 276.2327, Y 53.6800, Z -4.6667, A 0.000, B 0.000, C 0.000 }
gfCNCPoint3[22618] = {X 292.7731, Y 53.6800, Z -4.6667, A 0.000, B 0.000, C 0.000 }
gfCNCPoint3[22619] = {X 293.7344, Y 53.7883, Z -4.6667, A 0.000, B 0.000, C 0.000 }
gfCNCPoint3[22620] = {X 294.6475, Y 54.1078, Z -4.6667, A 0.000, B 0.000, C 0.000 }
gfCNCPoint3[22621] = {X 295.4666, Y 54.6225, Z -4.6667, A 0.000, B 0.000, C 0.000 }
gfCNCPoint3[22622] = {X 296.1506, Y 55.3065, Z -4.6667, A 0.000, B 0.000, C 0.000 }
gfCNCPoint3[22623] = {X 296.6653, Y 56.1256, Z -4.6667, A 0.000, B 0.000, C 0.000 }
gfCNCPoint3[22624] = {X 296.9848, Y 57.0387, Z -4.6667, A 0.000, B 0.000, C 0.000 }
gfCNCPoint3[22625] = {X 297.0931, Y 58.0000, Z -4.6667, A 0.000, B 0.000, C 0.000 }
gfCNCPoint3[22626] = {X 297.0931, Y 58.9351, Z -4.6667, A 0.000, B 0.000, C 0.000 }
gfCNCPoint3[22627] = {X 297.0008, Y 59.8116, Z -4.6667, A 0.000, B 0.000, C 0.000 }
gfCNCPoint3[22628] = {X 296.7332, Y 60.6513, Z -4.6667, A 0.000, B 0.000, C 0.000 }
gfCNCPoint3[22629] = {X 296.3014, Y 61.4196, Z -4.6667, A 0.000, B 0.000, C 0.000 }
gfCNCPoint3[22630] = {X 295.7231, Y 62.0847, Z -4.6667, A 0.000, B 0.000, C 0.000 }
gfCNCPoint3[22631] = {X 295.0223, Y 62.6191, Z -4.6667, A 0.000, B 0.000, C 0.000 }
gfCNCPoint3[22632] = {X 294.2279, Y 63.0009, Z -4.6667, A 0.000, B 0.000, C 0.000 }
gfCNCPoint3[22633] = {X 293.3728, Y 63.2141, Z -4.6667, A 0.000, B 0.000, C 0.000 }
gfCNCPoint3[22634] = {X 293.3845, Y 92.7811, Z -4.6667, A 0.000, B 0.000, C 0.000 }
gfCNCPoint3[22635] = {X 294.2370, Y 92.9986, Z -4.6667, A 0.000, B 0.000, C 0.000 }
gfCNCPoint3[22636] = {X 295.0284, Y 93.3831, Z -4.6667, A 0.000, B 0.000, C 0.000 }
gfCNCPoint3[22637] = {X 295.7263, Y 93.9188, Z -4.6667, A 0.000, B 0.000, C 0.000 }
gfCNCPoint3[22638] = {X 296.3022, Y 94.5840, Z -4.6667, A 0.000, B 0.000, C 0.000 }
gfCNCPoint3[22639] = {X 296.7326, Y 95.3514, Z -4.6667, A 0.000, B 0.000, C 0.000 }
gfCNCPoint3[22640] = {X 296.9998, Y 96.1896, Z -4.6667, A 0.000, B 0.000, C 0.000 }
gfCNCPoint3[22641] = {X 297.0931, Y 97.0645, Z -4.6667, A 0.000, B 0.000, C 0.000 }
gfCNCPoint3[22642] = {X 297.0931, Y 98.0000, Z -4.6667, A 0.000, B 0.000, C 0.000 }
gfCNCPoint3[22643] = {X 296.9848, Y 98.9613, Z -4.6667, A 0.000, B 0.000, C 0.000 }
gfCNCPoint3[22644] = {X 296.6653, Y 99.8744, Z -4.6667, A 0.000, B 0.000, C 0.000 }
gfCNCPoint3[22645] = {X 296.1506, Y 100.6935, Z -4.6667, A 0.000, B 0.000, C 0.000 }
gfCNCPoint3[22646] = {X 295.4666, Y 101.3775, Z -4.6667, A 0.000, B 0.000, C 0.000 }
gfCNCPoint3[22647] = {X 294.6475, Y 101.8922, Z -4.6667, A 0.000, B 0.000, C 0.000 }
gfCNCPoint3[22648] = {X 293.7344, Y 102.2117, Z -4.6667, A 0.000, B 0.000, C 0.000 }
gfCNCPoint3[22649] = {X 292.7731, Y 102.3200, Z -4.6667, A 0.000, B 0.000, C 0.000 }
gfCNCPoint3[22650] = {X 276.2327, Y 102.3200, Z -4.6667, A 0.000, B 0.000, C 0.000 }
gfCNCPoint3[22651] = {X 275.2714, Y 102.2117, Z -4.6667, A 0.000, B 0.000, C 0.000 }
gfCNCPoint3[22652] = {X 274.3583, Y 101.8922, Z -4.6667, A 0.000, B 0.000, C 0.000 }
gfCNCPoint3[22653] = {X 273.5392, Y 101.3775, Z -4.6667, A 0.000, B 0.000, C 0.000 }
gfCNCPoint3[22654] = {X 272.8552, Y 100.6935, Z -4.6667, A 0.000, B 0.000, C 0.000 }
gfCNCPoint3[22655] = {X 272.3405, Y 99.8744, Z -4.6667, A 0.000, B 0.000, C 0.000 }
gfCNCPoint3[22656] = {X 272.0210, Y 98.9613, Z -4.6667, A 0.000, B 0.000, C 0.000 }
gfCNCPoint3[22657] = {X 271.9127, Y 98.0000, Z -4.6667, A 0.000, B 0.000, C 0.000 }
gfCNCPoint3[22658] = {X 271.9127, Y 97.0659, Z -4.6667, A 0.000, B 0.000, C 0.000 }
gfCNCPoint3[22659] = {X 272.0026, Y 96.1891, Z -4.6667, A 0.000, B 0.000, C 0.000 }
gfCNCPoint3[22660] = {X 272.2686, Y 95.3488, Z -4.6667, A 0.000, B 0.000, C 0.000 }
gfCNCPoint3[22661] = {X 272.6996, Y 94.5800, Z -4.6667, A 0.000, B 0.000, C 0.000 }
gfCNCPoint3[22662] = {X 273.2777, Y 93.9146, Z -4.6667, A 0.000, B 0.000, C 0.000 }
gfCNCPoint3[22663] = {X 273.9788, Y 93.3805, Z -4.6667, A 0.000, B 0.000, C 0.000 }
gfCNCPoint3[22664] = {X 274.7737, Y 92.9997, Z -4.6667, A 0.000, B 0.000, C 0.000 }
gfCNCPoint3[22665] = {X 275.6294, Y 92.7883, Z -4.6667, A 0.000, B 0.000, C 0.000 }
gfCNCPoint3[22666] = {X 275.6294, Y 85.5950, Z -4.6667, A 0.000, B 0.000, C 0.000 }
gfCNCPoint3[22667] = {X 262.6397, Y 80.5030, Z -4.6667, A 0.000, B 0.000, C 0.000 }
gfCNCPoint3[22668] = {X 262.2771, Y 80.7316, Z -4.6667, A 0.000, B 0.000, C 0.000 }
gfCNCPoint3[22669] = {X 237.7967, Y 96.5881, Z -4.6667, A 0.000, B 0.000, C 0.000 }
gfCNCPoint3[22670] = {X 237.7998, Y 97.0649, Z -4.6667, A 0.000, B 0.000, C 0.000 }
gfCNCPoint3[22671] = {X 237.7998, Y 98.0000, Z -4.6667, A 0.000, B 0.000, C 0.000 }
gfCNCPoint3[22672] = {X 237.6915, Y 98.9613, Z -4.6667, A 0.000, B 0.000, C 0.000 }
gfCNCPoint3[22673] = {X 237.3720, Y 99.8744, Z -4.6667, A 0.000, B 0.000, C 0.000 }
gfCNCPoint3[22674] = {X 236.8573, Y 100.6935, Z -4.6667, A 0.000, B 0.000, C 0.000 }
gfCNCPoint3[22675] = {X 236.1733, Y 101.3775, Z -4.6667, A 0.000, B 0.000, C 0.000 }
gfCNCPoint3[22676] = {X 235.3542, Y 101.8922, Z -4.6667, A 0.000, B 0.000, C 0.000 }
gfCNCPoint3[22677] = {X 234.4411, Y 102.2117, Z -4.6667, A 0.000, B 0.000, C 0.000 }
gfCNCPoint3[22678] = {X 233.4798, Y 102.3200, Z -4.6667, A 0.000, B 0.000, C 0.000 }
gfCNCPoint3[22679] = {X 214.1790, Y 102.3200, Z -4.6667, A 0.000, B 0.000, C 0.000 }
gfCNCPoint3[22680] = {X 213.7862, Y 102.3021, Z -4.6667, A 0.000, B 0.000, C 0.000 }
gfCNCPoint3[22681] = {X 213.3966, Y 102.2485, Z -4.6667, A 0.000, B 0.000, C 0.000 }
gfCNCPoint3[22682] = {X 213.0070, Y 102.3021, Z -4.6667, A 0.000, B 0.000, C 0.000 }
gfCNCPoint3[22683] = {X 212.6141, Y 102.3200, Z -4.6667, A 0.000, B 0.000, C 0.000 }
gfCNCPoint3[22684] = {X 194.9870, Y 102.3200, Z -4.6667, A 0.000, B 0.000, C 0.000 }
gfCNCPoint3[22685] = {X 194.0257, Y 102.2117, Z -4.6667, A 0.000, B 0.000, C 0.000 }
gfCNCPoint3[22686] = {X 193.1126, Y 101.8922, Z -4.6667, A 0.000, B 0.000, C 0.000 }
gfCNCPoint3[22687] = {X 192.2935, Y 101.3775, Z -4.6667, A 0.000, B 0.000, C 0.000 }
gfCNCPoint3[22688] = {X 191.6094, Y 100.6935, Z -4.6667, A 0.000, B 0.000, C 0.000 }
gfCNCPoint3[22689] = {X 191.0948, Y 99.8744, Z -4.6667, A 0.000, B 0.000, C 0.000 }
gfCNCPoint3[22690] = {X 190.7753, Y 98.9613, Z -4.6667, A 0.000, B 0.000, C 0.000 }
gfCNCPoint3[22691] = {X 190.6670, Y 98.0000, Z -4.6667, A 0.000, B 0.000, C 0.000 }
gfCNCPoint3[22692] = {X 190.6670, Y 97.0659, Z -4.6667, A 0.000, B 0.000, C 0.000 }
gfCNCPoint3[22693] = {X 190.7727, Y 96.1162, Z -4.6667, A 0.000, B 0.000, C 0.000 }
gfCNCPoint3[22694] = {X 191.0846, Y 95.2129, Z -4.6667, A 0.000, B 0.000, C 0.000 }
gfCNCPoint3[22695] = {X 191.5874, Y 94.4003, Z -4.6667, A 0.000, B 0.000, C 0.000 }
gfCNCPoint3[22696] = {X 188.5647, Y 91.1002, Z -4.6667, A 0.000, B 0.000, C 0.000 }
gfCNCPoint3[22697] = {X 150.0898, Y 91.1002, Z -4.6667, A 0.000, B 0.000, C 0.000 }
gfCNCPoint3[22698] = {X 147.1450, Y 94.3628, Z -4.6667, A 0.000, B 0.000, C 0.000 }
gfCNCPoint3[22699] = {X 147.6638, Y 95.1840, Z -4.6667, A 0.000, B 0.000, C 0.000 }
gfCNCPoint3[22700] = {X 147.9872, Y 96.1000, Z -4.6667, A 0.000, B 0.000, C 0.000 }
gfCNCPoint3[22701] = {X 148.0991, Y 97.0650, Z -4.6667, A 0.000, B 0.000, C 0.000 }
gfCNCPoint3[22702] = {X 148.0991, Y 98.0000, Z -4.6667, A 0.000, B 0.000, C 0.000 }
gfCNCPoint3[22703] = {X 147.9908, Y 98.9613, Z -4.6667, A 0.000, B 0.000, C 0.000 }
gfCNCPoint3[22704] = {X 147.6713, Y 99.8744, Z -4.6667, A 0.000, B 0.000, C 0.000 }
gfCNCPoint3[22705] = {X 147.1566, Y 100.6935, Z -4.6667, A 0.000, B 0.000, C 0.000 }
gfCNCPoint3[22706] = {X 146.4726, Y 101.3775, Z -4.6667, A 0.000, B 0.000, C 0.000 }
gfCNCPoint3[22707] = {X 145.6535, Y 101.8922, Z -4.6667, A 0.000, B 0.000, C 0.000 }
gfCNCPoint3[22708] = {X 144.7404, Y 102.2117, Z -4.6667, A 0.000, B 0.000, C 0.000 }
gfCNCPoint3[22709] = {X 143.7791, Y 102.3200, Z -4.6667, A 0.000, B 0.000, C 0.000 }
gfCNCPoint3[22710] = {X 125.0000, Y 102.3200, Z -4.6667, A 0.000, B 0.000, C 0.000 }
gfCNCPoint3[22711] = {X 124.0387, Y 102.2117, Z -4.6667, A 0.000, B 0.000, C 0.000 }
gfCNCPoint3[22712] = {X 123.1256, Y 101.8922, Z -4.6667, A 0.000, B 0.000, C 0.000 }
gfCNCPoint3[22713] = {X 122.3065, Y 101.3775, Z -4.6667, A 0.000, B 0.000, C 0.000 }
gfCNCPoint3[22714] = {X 121.6225, Y 100.6935, Z -4.6667, A 0.000, B 0.000, C 0.000 }
gfCNCPoint3[22715] = {X 121.1078, Y 99.8744, Z -4.6667, A 0.000, B 0.000, C 0.000 }
gfCNCPoint3[22716] = {X 120.7883, Y 98.9613, Z -4.6667, A 0.000, B 0.000, C 0.000 }
gfCNCPoint3[22717] = {X 120.6800, Y 98.0000, Z -4.6667, A 0.000, B 0.000, C 0.000 }
gfCNCPoint3[22718] = {X 120.6800, Y 97.0659, Z -4.6667, A 0.000, B 0.000, C 0.000 }
gfCNCPoint3[22719] = {X 120.7832, Y 96.1273, Z -4.6667, A 0.000, B 0.000, C 0.000 }
gfCNCPoint3[22720] = {X 121.0879, Y 95.2336, Z -4.6667, A 0.000, B 0.000, C 0.000 }
gfCNCPoint3[22721] = {X 121.5794, Y 94.4273, Z -4.6667, A 0.000, B 0.000, C 0.000 }
gfCNCPoint3[22722] = {X 122.2345, Y 93.7472, Z -4.6667, A 0.000, B 0.000, C 0.000 }
gfCNCPoint3[22723] = {X 123.0216, Y 93.2256, Z -4.6667, A 0.000, B 0.000, C 0.000 }
gfCNCPoint3[22724] = {X 123.9032, Y 92.8875, Z -4.6667, A 0.000, B 0.000, C 0.000 }
gfCNCPoint3[22725] = {X 124.8373, Y 92.7490, Z -4.6667, A 0.000, B 0.000, C 0.000 }
gfCNCPoint3[22726] = {X 124.8816, Y 92.7319, Z -4.6667, A 0.000, B 0.000, C 0.000 }
gfCNCPoint3[22727] = {X 124.9279, Y 92.7215, Z -4.6667, A 0.000, B 0.000, C 0.000 }
gfCNCPoint3[22728] = {X 125.4494, Y 92.6441, Z -4.6667, A 0.000, B 0.000, C 0.000 }
gfCNCPoint3[22729] = {X 126.2806, Y 92.5043, Z -4.6667, A 0.000, B 0.000, C 0.000 }
gfCNCPoint3[22730] = {X 127.1002, Y 92.3078, Z -4.6667, A 0.000, B 0.000, C 0.000 }
gfCNCPoint3[22731] = {X 128.3217, Y 91.1564, Z -4.6667, A 0.000, B 0.000, C 0.000 }
gfCNCPoint3[22732] = {X 129.4789, Y 89.9402, Z -4.6667, A 0.000, B 0.000, C 0.000 }
gfCNCPoint3[22733] = {X 140.6802, Y 77.6397, Z -4.6667, A 0.000, B 0.000, C 0.000 }
gfCNCPoint3[22734] = {X 137.7227, Y 74.9465, Z -4.6667, A 0.000, B 0.000, C 0.000 }
gfCNCPoint3[22735] = {X 140.7393, Y 77.6936, Z -4.6667, A 0.000, B 0.000, C 0.000 }
gfCNCPoint3[22736] = {X 155.7327, Y 61.2289, Z -4.6667, A 0.000, B 0.000, C 0.000 }
gfCNCPoint3[22737] = {X 155.3668, Y 60.5226, Z -4.6667, A 0.000, B 0.000, C 0.000 }
gfCNCPoint3[22738] = {X 155.1393, Y 59.7604, Z -4.6667, A 0.000, B 0.000, C 0.000 }
gfCNCPoint3[22739] = {X 155.0581, Y 58.9691, Z -4.6667, A 0.000, B 0.000, C 0.000 }
gfCNCPoint3[22740] = {X 155.0580, Y 58.0000, Z -4.6667, A 0.000, B 0.000, C 0.000 }
gfCNCPoint3[22741] = {X 155.1643, Y 57.0565, Z -4.6667, A 0.000, B 0.000, C 0.000 }
gfCNCPoint3[22742] = {X 155.4778, Y 56.1603, Z -4.6667, A 0.000, B 0.000, C 0.000 }
gfCNCPoint3[22743] = {X 155.9830, Y 55.3564, Z -4.6667, A 0.000, B 0.000, C 0.000 }
gfCNCPoint3[22744] = {X 156.6544, Y 54.6850, Z -4.6667, A 0.000, B 0.000, C 0.000 }
gfCNCPoint3[22745] = {X 157.4583, Y 54.1799, Z -4.6667, A 0.000, B 0.000, C 0.000 }
gfCNCPoint3[22746] = {X 158.3545, Y 53.8663, Z -4.6667, A 0.000, B 0.000, C 0.000 }
gfCNCPoint3[22747] = {X 159.2980, Y 53.7600, Z -4.6667, A 0.000, B 0.000, C 0.000 }
gfCNCPoint3[22748] = {X 178.5335, Y 53.7600, Z -4.6667, A 0.000, B 0.000, C 0.000 }
gfCNCPoint3[22749] = {X 179.4770, Y 53.8663, Z -4.6667, A 0.000, B 0.000, C 0.000 }
gfCNCPoint3[22750] = {X 180.3732, Y 54.1799, Z -4.6667, A 0.000, B 0.000, C 0.000 }
gfCNCPoint3[22751] = {X 181.1771, Y 54.6850, Z -4.6667, A 0.000, B 0.000, C 0.000 }
gfCNCPoint3[22752] = {X 181.8485, Y 55.3564, Z -4.6667, A 0.000, B 0.000, C 0.000 }
gfCNCPoint3[22753] = {X 182.3536, Y 56.1603, Z -4.6667, A 0.000, B 0.000, C 0.000 }
gfCNCPoint3[22754] = {X 182.6672, Y 57.0565, Z -4.6667, A 0.000, B 0.000, C 0.000 }
gfCNCPoint3[22755] = {X 182.7735, Y 58.0000, Z -4.6667, A 0.000, B 0.000, C 0.000 }
gfCNCPoint3[22756] = {X 182.7735, Y 58.9342, Z -4.6667, A 0.000, B 0.000, C 0.000 }
gfCNCPoint3[22757] = {X 182.6984, Y 59.7284, Z -4.6667, A 0.000, B 0.000, C 0.000 }
gfCNCPoint3[22758] = {X 182.4759, Y 60.4945, Z -4.6667, A 0.000, B 0.000, C 0.000 }
gfCNCPoint3[22759] = {X 182.1139, Y 61.2053, Z -4.6667, A 0.000, B 0.000, C 0.000 }
gfCNCPoint3[22760] = {X 209.4198, Y 91.0082, Z -4.6667, A 0.000, B 0.000, C 0.000 }
gfCNCPoint3[22761] = {X 210.0810, Y 91.6791, Z -4.6667, A 0.000, B 0.000, C 0.000 }
gfCNCPoint3[22762] = {X 210.7893, Y 92.3000, Z -4.6667, A 0.000, B 0.000, C 0.000 }
gfCNCPoint3[22763] = {X 211.0804, Y 92.4840, Z -4.6667, A 0.000, B 0.000, C 0.000 }
gfCNCPoint3[22764] = {X 211.4067, Y 92.5940, Z -4.6667, A 0.000, B 0.000, C 0.000 }
gfCNCPoint3[22765] = {X 213.4017, Y 92.9051, Z -4.6667, A 0.000, B 0.000, C 0.000 }
gfCNCPoint3[22766] = {X 214.4546, Y 92.8160, Z -4.6667, A 0.000, B 0.000, C 0.000 }
gfCNCPoint3[22767] = {X 215.5096, Y 92.7555, Z -4.6667, A 0.000, B 0.000, C 0.000 }
gfCNCPoint3[22768] = {X 216.1941, Y 92.6806, Z -4.6667, A 0.000, B 0.000, C 0.000 }
gfCNCPoint3[22769] = {X 216.8531, Y 92.4813, Z -4.6667, A 0.000, B 0.000, C 0.000 }
gfCNCPoint3[22770] = {X 217.4643, Y 92.1643, Z -4.6667, A 0.000, B 0.000, C 0.000 }
gfCNCPoint3[22771] = {X 223.0046, Y 88.5889, Z -4.6667, A 0.000, B 0.000, C 0.000 }
gfCNCPoint3[22772] = {X 246.0034, Y 73.8824, Z -4.6667, A 0.000, B 0.000, C 0.000 }
gfCNCPoint3[22773] = {X 221.6602, Y 64.3294, Z -4.6667, A 0.000, B 0.000, C 0.000 }
gfCNCPoint3[22774] = {X 219.8841, Y 63.7349, Z -4.6667, A 0.000, B 0.000, C 0.000 }
gfCNCPoint3[22775] = {X 218.0518, Y 63.3473, Z -4.6667, A 0.000, B 0.000, C 0.000 }
gfCNCPoint3[22776] = {X 216.1871, Y 63.1716, Z -4.6667, A 0.000, B 0.000, C 0.000 }
gfCNCPoint3[22777] = {X 215.2724, Y 63.0398, Z -4.6667, A 0.000, B 0.000, C 0.000 }
gfCNCPoint3[22778] = {X 214.4081, Y 62.7130, Z -4.6667, A 0.000, B 0.000, C 0.000 }
gfCNCPoint3[22779] = {X 213.6350, Y 62.2067, Z -4.6667, A 0.000, B 0.000, C 0.000 }
gfCNCPoint3[22780] = {X 212.9901, Y 61.5450, Z -4.6667, A 0.000, B 0.000, C 0.000 }
gfCNCPoint3[22781] = {X 212.5038, Y 60.7592, Z -4.6667, A 0.000, B 0.000, C 0.000 }
gfCNCPoint3[22782] = {X 212.1992, Y 59.8868, Z -4.6667, A 0.000, B 0.000, C 0.000 }
gfCNCPoint3[22783] = {X 212.0910, Y 58.9691, Z -4.6667, A 0.000, B 0.000, C 0.000 }
gfCNCPoint3[22784] = {X 212.0908, Y 58.0000, Z -4.6667, A 0.000, B 0.000, C 0.000 }
gfCNCPoint3[22785] = {X 212.1971, Y 57.0565, Z -4.6667, A 0.000, B 0.000, C 0.000 }
gfCNCPoint3[22786] = {X 212.5107, Y 56.1603, Z -4.6667, A 0.000, B 0.000, C 0.000 }
gfCNCPoint3[22787] = {X 213.0158, Y 55.3564, Z -4.6667, A 0.000, B 0.000, C 0.000 }
gfCNCPoint3[22788] = {X 213.6872, Y 54.6850, Z -4.6667, A 0.000, B 0.000, C 0.000 }
gfCNCPoint3[22789] = {X 214.4911, Y 54.1799, Z -4.6667, A 0.000, B 0.000, C 0.000 }
gfCNCPoint3[22790] = {X 215.3873, Y 53.8663, Z -4.6667, A 0.000, B 0.000, C 0.000 }
gfCNCPoint3[22791] = {X 216.3308, Y 53.7600, Z -4.6667, A 0.000, B 0.000, C 0.000 }
gfCNCPoint3[22792] = {X 237.2617, Y 53.7600, Z -4.6667, A 0.000, B 0.000, C 0.000 }
gfCNCPoint3[22793] = {X 238.2052, Y 53.8663, Z -4.6667, A 0.000, B 0.000, C 0.000 }
gfCNCPoint3[22794] = {X 239.1014, Y 54.1799, Z -4.6667, A 0.000, B 0.000, C 0.000 }
gfCNCPoint3[22795] = {X 239.9053, Y 54.6850, Z -4.6667, A 0.000, B 0.000, C 0.000 }
gfCNCPoint3[22796] = {X 240.5767, Y 55.3564, Z -4.6667, A 0.000, B 0.000, C 0.000 }
gfCNCPoint3[22797] = {X 241.0818, Y 56.1603, Z -4.6667, A 0.000, B 0.000, C 0.000 }
gfCNCPoint3[22798] = {X 241.3954, Y 57.0565, Z -4.6667, A 0.000, B 0.000, C 0.000 }
gfCNCPoint3[22799] = {X 241.5017, Y 58.0000, Z -4.6667, A 0.000, B 0.000, C 0.000 }
gfCNCPoint3[22800] = {X 241.5017, Y 58.2870, Z -4.6667, A 0.000, B 0.000, C 0.000 }
gfCNCPoint3[22801] = {X 248.0845, Y 60.8537, Z -4.6667, A 0.000, B 0.000, C 0.000 }
gfCNCPoint3[22802] = {X 275.7128, Y 71.8199, Z -4.6667, A 0.000, B 0.000, C 0.000 }
gfCNCPoint3[22803] = {X 275.7140, Y 63.1422, Z -4.6667, A 0.000, B 0.000, C 0.000 }
gfCNCPoint3[22804] = {X 274.8654, Y 62.9476, Z -4.6667, A 0.000, B 0.000, C 0.000 }
gfCNCPoint3[22805] = {X 274.0744, Y 62.5837, Z -4.6667, A 0.000, B 0.000, C 0.000 }
gfCNCPoint3[22806] = {X 273.3745, Y 62.0659, Z -4.6667, A 0.000, B 0.000, C 0.000 }
gfCNCPoint3[22807] = {X 272.7951, Y 61.4161, Z -4.6667, A 0.000, B 0.000, C 0.000 }
gfCNCPoint3[22808] = {X 272.3606, Y 60.6616, Z -4.6667, A 0.000, B 0.000, C 0.000 }
gfCNCPoint3[22809] = {X 272.0894, Y 59.8343, Z -4.6667, A 0.000, B 0.000, C 0.000 }
gfCNCPoint3[22810] = {X 271.9928, Y 58.9691, Z -4.6667, A 0.000, B 0.000, C 0.000 }
gfCNCPoint3[22811] = {X 271.9927, Y 58.0000, Z -4.6667, A 0.000, B 0.000, C 0.000 }
gfCNCPoint3[22812] = {X 272.0990, Y 57.0565, Z -4.6667, A 0.000, B 0.000, C 0.000 }
gfCNCPoint3[22813] = {X 272.4126, Y 56.1603, Z -4.6667, A 0.000, B 0.000, C 0.000 }
gfCNCPoint3[22814] = {X 272.9177, Y 55.3564, Z -4.6667, A 0.000, B 0.000, C 0.000 }
gfCNCPoint3[22815] = {X 273.5891, Y 54.6850, Z -4.6667, A 0.000, B 0.000, C 0.000 }
gfCNCPoint3[22816] = {X 274.3930, Y 54.1799, Z -4.6667, A 0.000, B 0.000, C 0.000 }
gfCNCPoint3[22817] = {X 275.2892, Y 53.8663, Z -4.6667, A 0.000, B 0.000, C 0.000 }
gfCNCPoint3[22818] = {X 276.2327, Y 53.7600, Z -4.6667, A 0.000, B 0.000, C 0.000 }
gfCNCPoint3[22819] = {X 292.7731, Y 53.7600, Z -4.6667, A 0.000, B 0.000, C 0.000 }
